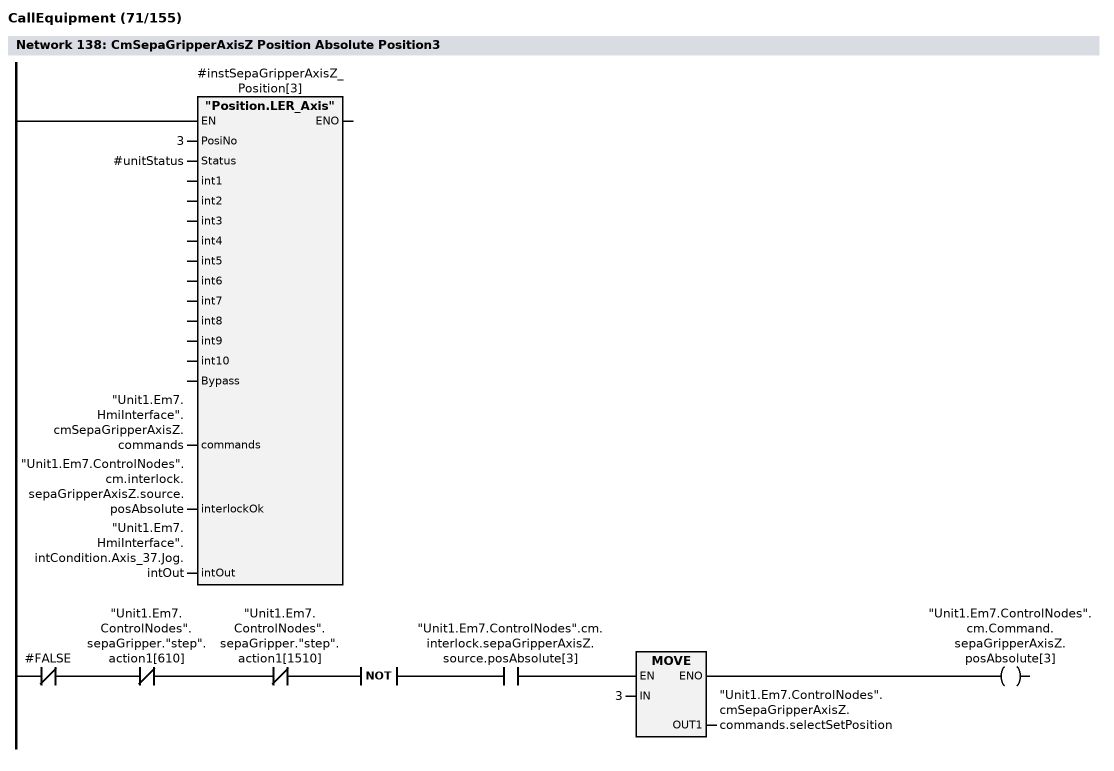
   RUNG wire#powerrail
      #instSepaGripperAxisZ_Position[3](PosiNo := 3, Status := #unitStatus, int1 :=, int2 :=, int3 :=, int4 :=, int5 :=, int6 :=, int7 :=, int8 :=, int9 :=, int10 :=, Bypass :=, commands := "Unit1.Em7.HmiInterface".cmSepaGripperAxisZ.commands, interlockOk := "Unit1.Em7.ControlNodes".cm.interlock.sepaGripperAxisZ.source.posAbsolute, intOut := "Unit1.Em7.HmiInterface".intCondition.Axis_37.Jog.intOut)
   END_RUNG
   RUNG wire#powerrail
      I_Contact( #FALSE )
      I_Contact( "Unit1.Em7.ControlNodes".sepaGripper."step".action1[610] )
      I_Contact( "Unit1.Em7.ControlNodes".sepaGripper."step".action1[1510] )
      Not()
      Contact( "Unit1.Em7.ControlNodes".cm.interlock.sepaGripperAxisZ.source.posAbsolute[3] )
      Move(in := 3, out1 => "Unit1.Em7.ControlNodes".cmSepaGripperAxisZ.commands.selectSetPosition)
      Coil( "Unit1.Em7.ControlNodes".cm.Command.sepaGripperAxisZ.posAbsolute[3] )
   END_RUNG
   // the same network as SCL:
   #instSepaGripperAxisZ_Position[3](PosiNo := 3,   // "Position.LER_Axis"
                           Status := #unitStatus,
                           commands := "Unit1.Em7.HmiInterface".cmSepaGripperAxisZ.commands,
                           interlockOk := "Unit1.Em7.ControlNodes".cm.interlock.sepaGripperAxisZ.source.posAbsolute,
                           intOut := "Unit1.Em7.HmiInterface".intCondition.Axis_37.Jog.intOut);
   #_w1 := NOT (NOT #FALSE AND NOT "Unit1.Em7.ControlNodes".sepaGripper."step".action1[610] AND NOT "Unit1.Em7.ControlNodes".sepaGripper."step".action1[1510]) AND "Unit1.Em7.ControlNodes".cm.interlock.sepaGripperAxisZ.source.posAbsolute[3];
   IF #_w1 THEN "Unit1.Em7.ControlNodes".cmSepaGripperAxisZ.commands.selectSetPosition := 3; END_IF;
   "Unit1.Em7.ControlNodes".cm.Command.sepaGripperAxisZ.posAbsolute[3] := #_w1;
END_REGION

REGION Network 139: CmSepaGripperAxisZ Position Absolute Position4
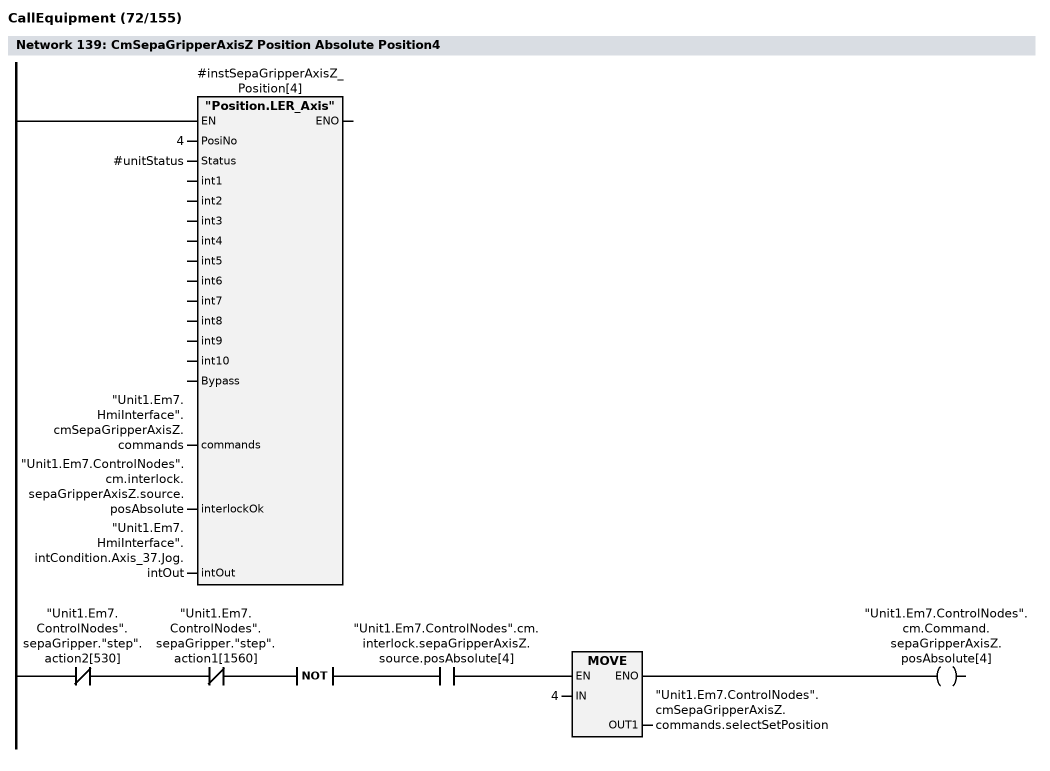
   RUNG wire#powerrail
      #instSepaGripperAxisZ_Position[4](PosiNo := 4, Status := #unitStatus, int1 :=, int2 :=, int3 :=, int4 :=, int5 :=, int6 :=, int7 :=, int8 :=, int9 :=, int10 :=, Bypass :=, commands := "Unit1.Em7.HmiInterface".cmSepaGripperAxisZ.commands, interlockOk := "Unit1.Em7.ControlNodes".cm.interlock.sepaGripperAxisZ.source.posAbsolute, intOut := "Unit1.Em7.HmiInterface".intCondition.Axis_37.Jog.intOut)
   END_RUNG
   RUNG wire#powerrail
      I_Contact( "Unit1.Em7.ControlNodes".sepaGripper."step".action2[530] )
      I_Contact( "Unit1.Em7.ControlNodes".sepaGripper."step".action1[1560] )
      Not()
      Contact( "Unit1.Em7.ControlNodes".cm.interlock.sepaGripperAxisZ.source.posAbsolute[4] )
      Move(in := 4, out1 => "Unit1.Em7.ControlNodes".cmSepaGripperAxisZ.commands.selectSetPosition)
      Coil( "Unit1.Em7.ControlNodes".cm.Command.sepaGripperAxisZ.posAbsolute[4] )
   END_RUNG
   // the same network as SCL:
   #instSepaGripperAxisZ_Position[4](PosiNo := 4,   // "Position.LER_Axis"
                           Status := #unitStatus,
                           commands := "Unit1.Em7.HmiInterface".cmSepaGripperAxisZ.commands,
                           interlockOk := "Unit1.Em7.ControlNodes".cm.interlock.sepaGripperAxisZ.source.posAbsolute,
                           intOut := "Unit1.Em7.HmiInterface".intCondition.Axis_37.Jog.intOut);
   #_w1 := NOT (NOT "Unit1.Em7.ControlNodes".sepaGripper."step".action2[530] AND NOT "Unit1.Em7.ControlNodes".sepaGripper."step".action1[1560]) AND "Unit1.Em7.ControlNodes".cm.interlock.sepaGripperAxisZ.source.posAbsolute[4];
   IF #_w1 THEN "Unit1.Em7.ControlNodes".cmSepaGripperAxisZ.commands.selectSetPosition := 4; END_IF;
   "Unit1.Em7.ControlNodes".cm.Command.sepaGripperAxisZ.posAbsolute[4] := #_w1;
END_REGION

REGION Network 140: CmSepaGripperAxisZ Position Absolute Position5
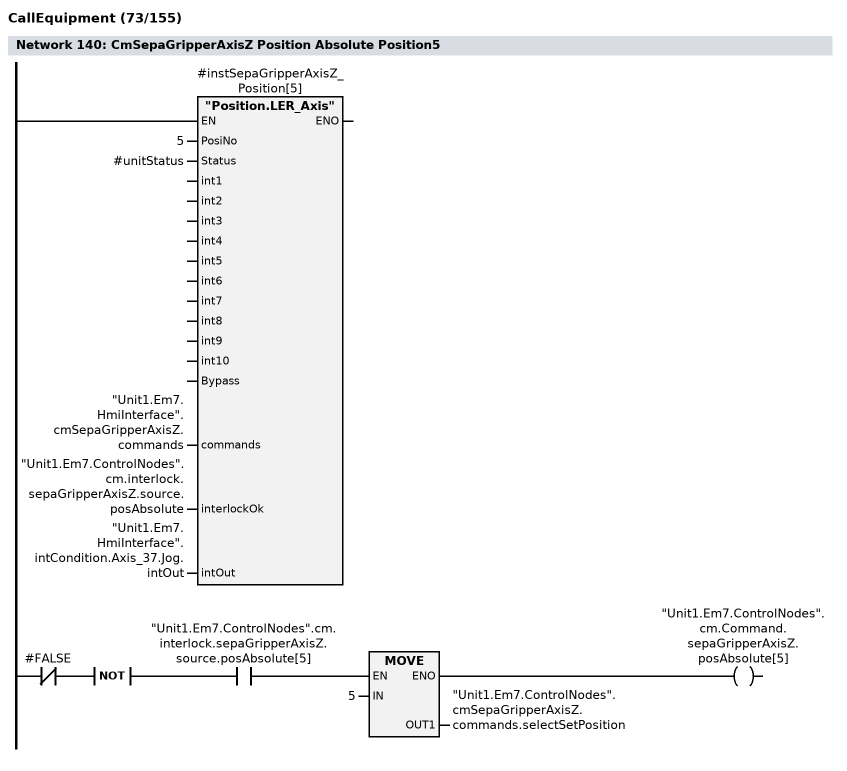
   RUNG wire#powerrail
      #instSepaGripperAxisZ_Position[5](PosiNo := 5, Status := #unitStatus, int1 :=, int2 :=, int3 :=, int4 :=, int5 :=, int6 :=, int7 :=, int8 :=, int9 :=, int10 :=, Bypass :=, commands := "Unit1.Em7.HmiInterface".cmSepaGripperAxisZ.commands, interlockOk := "Unit1.Em7.ControlNodes".cm.interlock.sepaGripperAxisZ.source.posAbsolute, intOut := "Unit1.Em7.HmiInterface".intCondition.Axis_37.Jog.intOut)
   END_RUNG
   RUNG wire#powerrail
      I_Contact( #FALSE )
      Not()
      Contact( "Unit1.Em7.ControlNodes".cm.interlock.sepaGripperAxisZ.source.posAbsolute[5] )
      Move(in := 5, out1 => "Unit1.Em7.ControlNodes".cmSepaGripperAxisZ.commands.selectSetPosition)
      Coil( "Unit1.Em7.ControlNodes".cm.Command.sepaGripperAxisZ.posAbsolute[5] )
   END_RUNG
   // the same network as SCL:
   #instSepaGripperAxisZ_Position[5](PosiNo := 5,   // "Position.LER_Axis"
                           Status := #unitStatus,
                           commands := "Unit1.Em7.HmiInterface".cmSepaGripperAxisZ.commands,
                           interlockOk := "Unit1.Em7.ControlNodes".cm.interlock.sepaGripperAxisZ.source.posAbsolute,
                           intOut := "Unit1.Em7.HmiInterface".intCondition.Axis_37.Jog.intOut);
   #_w1 := NOT (NOT #FALSE) AND "Unit1.Em7.ControlNodes".cm.interlock.sepaGripperAxisZ.source.posAbsolute[5];
   IF #_w1 THEN "Unit1.Em7.ControlNodes".cmSepaGripperAxisZ.commands.selectSetPosition := 5; END_IF;
   "Unit1.Em7.ControlNodes".cm.Command.sepaGripperAxisZ.posAbsolute[5] := #_w1;
END_REGION

REGION Network 141: CmSepaGripperAxisZ Position Absolute Position6
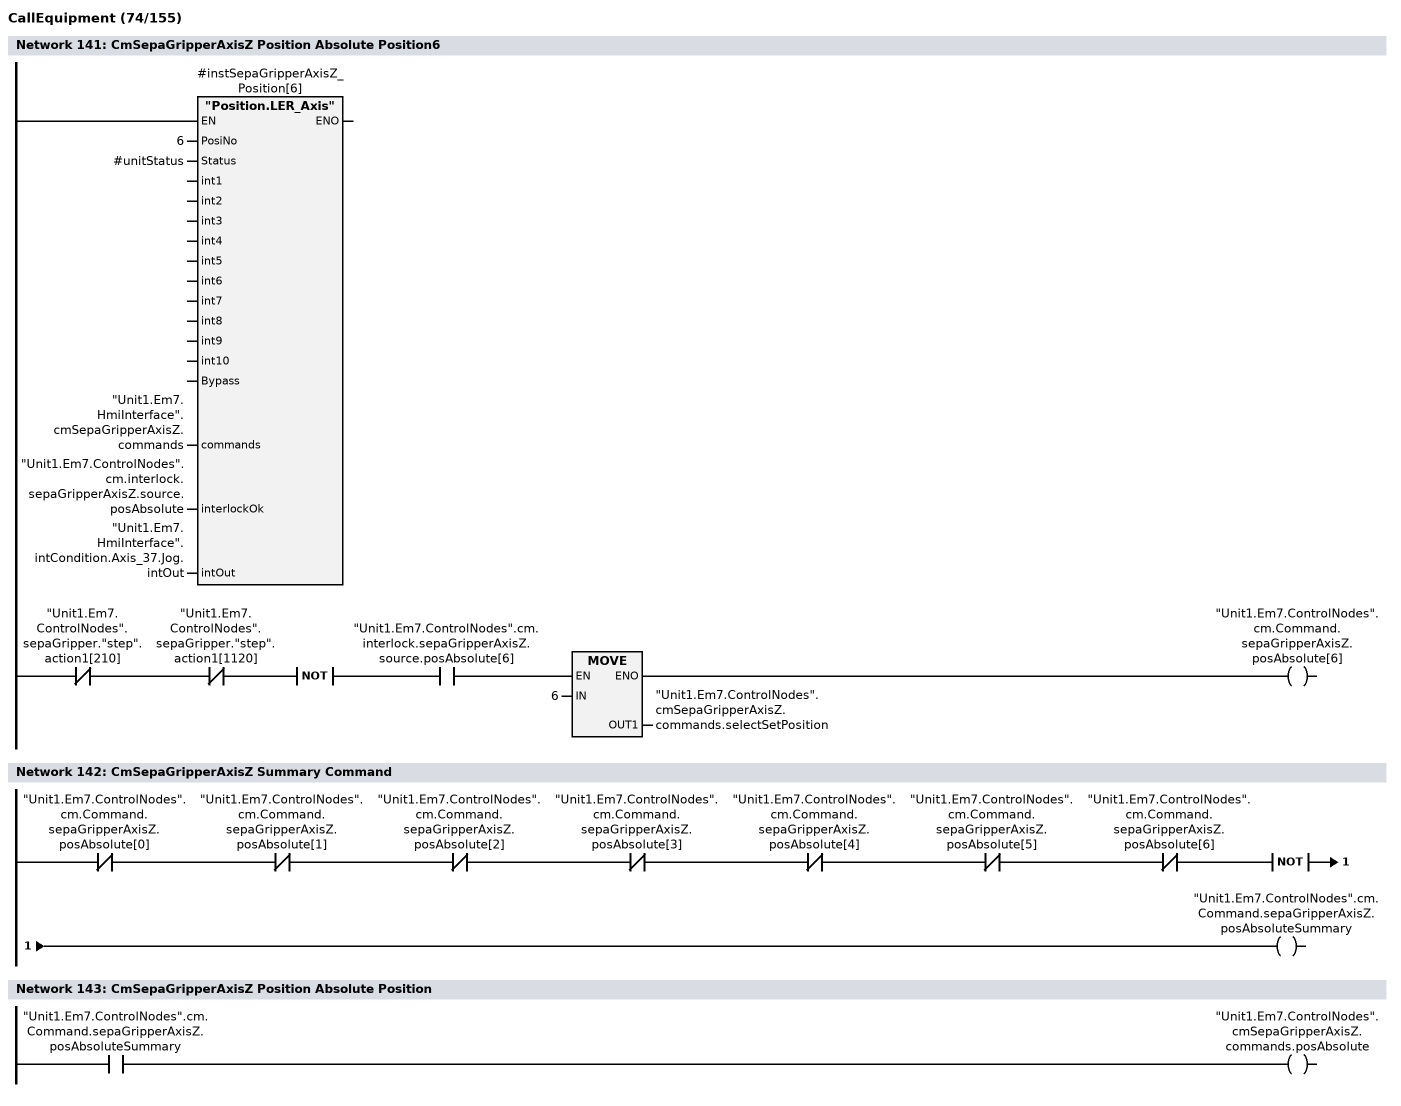
   RUNG wire#powerrail
      #instSepaGripperAxisZ_Position[6](PosiNo := 6, Status := #unitStatus, int1 :=, int2 :=, int3 :=, int4 :=, int5 :=, int6 :=, int7 :=, int8 :=, int9 :=, int10 :=, Bypass :=, commands := "Unit1.Em7.HmiInterface".cmSepaGripperAxisZ.commands, interlockOk := "Unit1.Em7.ControlNodes".cm.interlock.sepaGripperAxisZ.source.posAbsolute, intOut := "Unit1.Em7.HmiInterface".intCondition.Axis_37.Jog.intOut)
   END_RUNG
   RUNG wire#powerrail
      I_Contact( "Unit1.Em7.ControlNodes".sepaGripper."step".action1[210] )
      I_Contact( "Unit1.Em7.ControlNodes".sepaGripper."step".action1[1120] )
      Not()
      Contact( "Unit1.Em7.ControlNodes".cm.interlock.sepaGripperAxisZ.source.posAbsolute[6] )
      Move(in := 6, out1 => "Unit1.Em7.ControlNodes".cmSepaGripperAxisZ.commands.selectSetPosition)
      Coil( "Unit1.Em7.ControlNodes".cm.Command.sepaGripperAxisZ.posAbsolute[6] )
   END_RUNG
   // the same network as SCL:
   #instSepaGripperAxisZ_Position[6](PosiNo := 6,   // "Position.LER_Axis"
                           Status := #unitStatus,
                           commands := "Unit1.Em7.HmiInterface".cmSepaGripperAxisZ.commands,
                           interlockOk := "Unit1.Em7.ControlNodes".cm.interlock.sepaGripperAxisZ.source.posAbsolute,
                           intOut := "Unit1.Em7.HmiInterface".intCondition.Axis_37.Jog.intOut);
   #_w1 := NOT (NOT "Unit1.Em7.ControlNodes".sepaGripper."step".action1[210] AND NOT "Unit1.Em7.ControlNodes".sepaGripper."step".action1[1120]) AND "Unit1.Em7.ControlNodes".cm.interlock.sepaGripperAxisZ.source.posAbsolute[6];
   IF #_w1 THEN "Unit1.Em7.ControlNodes".cmSepaGripperAxisZ.commands.selectSetPosition := 6; END_IF;
   "Unit1.Em7.ControlNodes".cm.Command.sepaGripperAxisZ.posAbsolute[6] := #_w1;
END_REGION

REGION Network 142: CmSepaGripperAxisZ Summary Command
   RUNG wire#powerrail
      I_Contact( "Unit1.Em7.ControlNodes".cm.Command.sepaGripperAxisZ.posAbsolute[0] )
      I_Contact( "Unit1.Em7.ControlNodes".cm.Command.sepaGripperAxisZ.posAbsolute[1] )
      I_Contact( "Unit1.Em7.ControlNodes".cm.Command.sepaGripperAxisZ.posAbsolute[2] )
      I_Contact( "Unit1.Em7.ControlNodes".cm.Command.sepaGripperAxisZ.posAbsolute[3] )
      I_Contact( "Unit1.Em7.ControlNodes".cm.Command.sepaGripperAxisZ.posAbsolute[4] )
      I_Contact( "Unit1.Em7.ControlNodes".cm.Command.sepaGripperAxisZ.posAbsolute[5] )
      I_Contact( "Unit1.Em7.ControlNodes".cm.Command.sepaGripperAxisZ.posAbsolute[6] )
      Not()
      Coil( "Unit1.Em7.ControlNodes".cm.Command.sepaGripperAxisZ.posAbsoluteSummary )
   END_RUNG
   // the same network as SCL:
   "Unit1.Em7.ControlNodes".cm.Command.sepaGripperAxisZ.posAbsoluteSummary := NOT (NOT "Unit1.Em7.ControlNodes".cm.Command.sepaGripperAxisZ.posAbsolute[0] AND NOT "Unit1.Em7.ControlNodes".cm.Command.sepaGripperAxisZ.posAbsolute[1] AND NOT "Unit1.Em7.ControlNodes".cm.Command.sepaGripperAxisZ.posAbsolute[2] AND NOT "Unit1.Em7.ControlNodes".cm.Command.sepaGripperAxisZ.posAbsolute[3] AND NOT "Unit1.Em7.ControlNodes".cm.Command.sepaGripperAxisZ.posAbsolute[4] AND NOT "Unit1.Em7.ControlNodes".cm.Command.sepaGripperAxisZ.posAbsolute[5] AND NOT "Unit1.Em7.ControlNodes".cm.Command.sepaGripperAxisZ.posAbsolute[6]);
END_REGION

REGION Network 143: CmSepaGripperAxisZ Position Absolute Position
   RUNG wire#powerrail
      Contact( "Unit1.Em7.ControlNodes".cm.Command.sepaGripperAxisZ.posAbsoluteSummary )
      Coil( "Unit1.Em7.ControlNodes".cmSepaGripperAxisZ.commands.posAbsolute )
   END_RUNG
   // the same network as SCL:
   "Unit1.Em7.ControlNodes".cmSepaGripperAxisZ.commands.posAbsolute := "Unit1.Em7.ControlNodes".cm.Command.sepaGripperAxisZ.posAbsoluteSummary;
END_REGION

REGION Network 144: CmSepaGripperAxisZ Interlock Summary
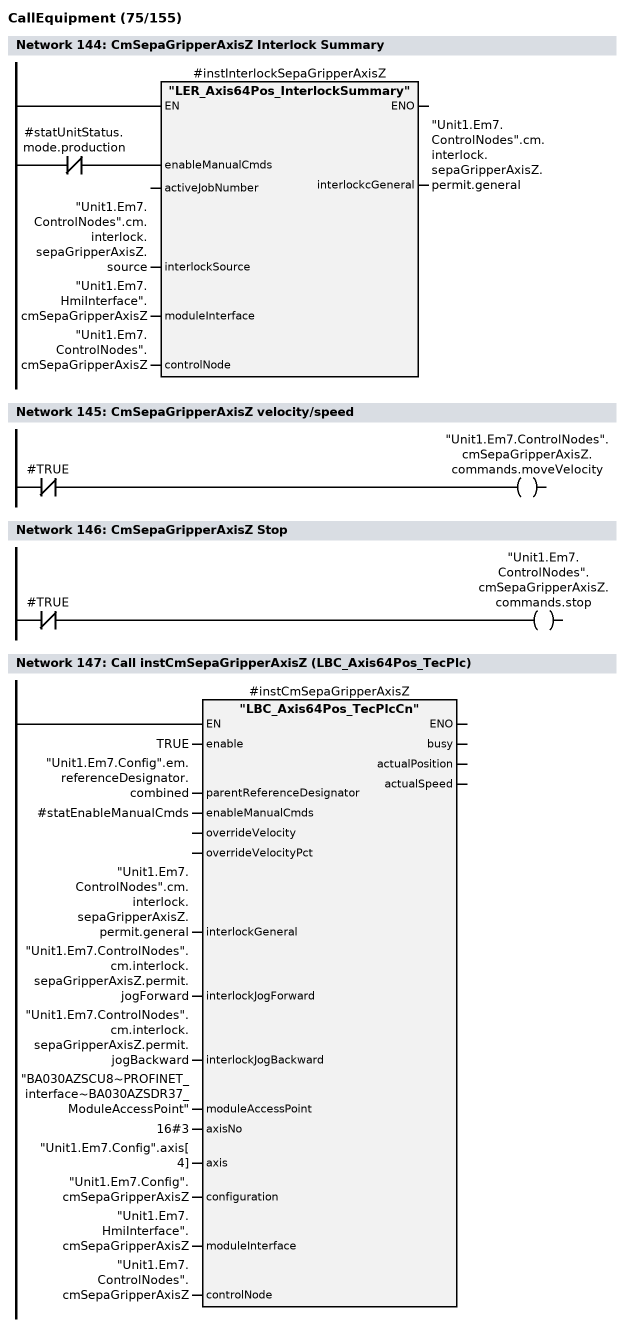
   RUNG wire#powerrail
      #instInterlockSepaGripperAxisZ(enableManualCmds := wire#w1, activeJobNumber :=, interlockSource := "Unit1.Em7.ControlNodes".cm.interlock.sepaGripperAxisZ.source, moduleInterface := "Unit1.Em7.HmiInterface".cmSepaGripperAxisZ, controlNode := "Unit1.Em7.ControlNodes".cmSepaGripperAxisZ, interlockcGeneral => "Unit1.Em7.ControlNodes".cm.interlock.sepaGripperAxisZ.permit.general)
   END_RUNG
   RUNG wire#powerrail
      I_Contact( #statUnitStatus.mode.production )
   END_RUNG wire#w1
   // the same network as SCL:
   #instInterlockSepaGripperAxisZ(enableManualCmds := NOT #statUnitStatus.mode.production,   // "LER_Axis64Pos_InterlockSummary"
                           interlockSource := "Unit1.Em7.ControlNodes".cm.interlock.sepaGripperAxisZ.source,
                           moduleInterface := "Unit1.Em7.HmiInterface".cmSepaGripperAxisZ,
                           controlNode := "Unit1.Em7.ControlNodes".cmSepaGripperAxisZ,
                           interlockcGeneral => "Unit1.Em7.ControlNodes".cm.interlock.sepaGripperAxisZ.permit.general);
END_REGION

REGION Network 145: CmSepaGripperAxisZ velocity/speed
   RUNG wire#powerrail
      I_Contact( #TRUE )
      Coil( "Unit1.Em7.ControlNodes".cmSepaGripperAxisZ.commands.moveVelocity )
   END_RUNG
   // the same network as SCL:
   "Unit1.Em7.ControlNodes".cmSepaGripperAxisZ.commands.moveVelocity := NOT #TRUE;
END_REGION

REGION Network 146: CmSepaGripperAxisZ Stop
   RUNG wire#powerrail
      I_Contact( #TRUE )
      Coil( "Unit1.Em7.ControlNodes".cmSepaGripperAxisZ.commands.stop )
   END_RUNG
   // the same network as SCL:
   "Unit1.Em7.ControlNodes".cmSepaGripperAxisZ.commands.stop := NOT #TRUE;
END_REGION

REGION Network 147: Call instCmSepaGripperAxisZ (LBC_Axis64Pos_TecPlc)
   RUNG wire#powerrail
      #instCmSepaGripperAxisZ(enable := TRUE, parentReferenceDesignator := "Unit1.Em7.Config".em.referenceDesignator.combined, enableManualCmds := #statEnableManualCmds, overrideVelocity :=, overrideVelocityPct :=, interlockGeneral := "Unit1.Em7.ControlNodes".cm.interlock.sepaGripperAxisZ.permit.general, interlockJogForward := "Unit1.Em7.ControlNodes".cm.interlock.sepaGripperAxisZ.permit.jogForward, interlockJogBackward := "Unit1.Em7.ControlNodes".cm.interlock.sepaGripperAxisZ.permit.jogBackward, moduleAccessPoint := "BA030AZSCU8~PROFINET_interface~BA030AZSDR37_ModuleAccessPoint", axisNo := 16#3, axis := "Unit1.Em7.Config".axis[4], configuration := "Unit1.Em7.Config".cmSepaGripperAxisZ, moduleInterface := "Unit1.Em7.HmiInterface".cmSepaGripperAxisZ, controlNode := "Unit1.Em7.ControlNodes".cmSepaGripperAxisZ, busy =>, actualPosition =>, actualSpeed =>)
   END_RUNG
   // the same network as SCL:
   #instCmSepaGripperAxisZ(enable := TRUE,   // "LBC_Axis64Pos_TecPlcCn"
                           parentReferenceDesignator := "Unit1.Em7.Config".em.referenceDesignator.combined,
                           enableManualCmds := #statEnableManualCmds,
                           interlockGeneral := "Unit1.Em7.ControlNodes".cm.interlock.sepaGripperAxisZ.permit.general,
                           interlockJogForward := "Unit1.Em7.ControlNodes".cm.interlock.sepaGripperAxisZ.permit.jogForward,
                           interlockJogBackward := "Unit1.Em7.ControlNodes".cm.interlock.sepaGripperAxisZ.permit.jogBackward,
                           moduleAccessPoint := "BA030AZSCU8~PROFINET_interface~BA030AZSDR37_ModuleAccessPoint",
                           axisNo := 16#3,
                           axis := "Unit1.Em7.Config".axis[4],
                           configuration := "Unit1.Em7.Config".cmSepaGripperAxisZ,
                           moduleInterface := "Unit1.Em7.HmiInterface".cmSepaGripperAxisZ,
                           controlNode := "Unit1.Em7.ControlNodes".cmSepaGripperAxisZ);
END_REGION

REGION Network 148: CmSepaGripperAxisZ SoftCam
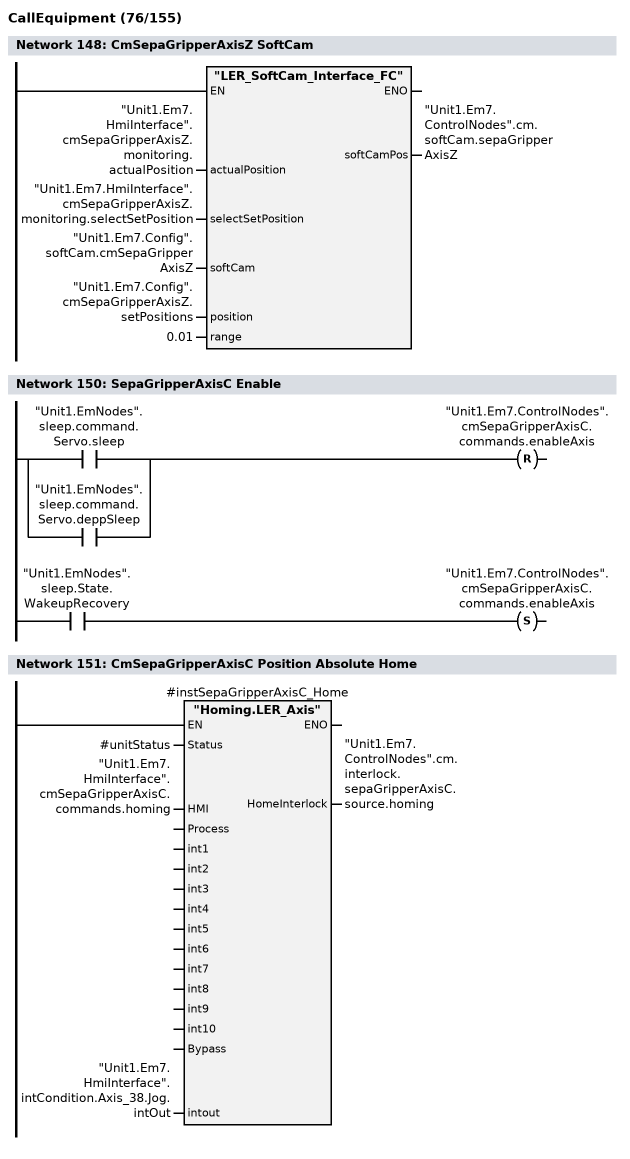
   RUNG wire#powerrail
      "LER_SoftCam_Interface_FC"(actualPosition := "Unit1.Em7.HmiInterface".cmSepaGripperAxisZ.monitoring.actualPosition, selectSetPosition := "Unit1.Em7.HmiInterface".cmSepaGripperAxisZ.monitoring.selectSetPosition, softCam := "Unit1.Em7.Config".softCam.cmSepaGripperAxisZ, position := "Unit1.Em7.Config".cmSepaGripperAxisZ.setPositions, range := 0.01, softCamPos => "Unit1.Em7.ControlNodes".cm.softCam.sepaGripperAxisZ)
   END_RUNG
   // the same network as SCL:
   "LER_SoftCam_Interface_FC"(actualPosition := "Unit1.Em7.HmiInterface".cmSepaGripperAxisZ.monitoring.actualPosition,
                           selectSetPosition := "Unit1.Em7.HmiInterface".cmSepaGripperAxisZ.monitoring.selectSetPosition,
                           softCam := "Unit1.Em7.Config".softCam.cmSepaGripperAxisZ,
                           position := "Unit1.Em7.Config".cmSepaGripperAxisZ.setPositions,
                           range := 0.01,
                           softCamPos => "Unit1.Em7.ControlNodes".cm.softCam.sepaGripperAxisZ);
END_REGION

REGION Network 150: SepaGripperAxisC Enable
   RUNG wire#powerrail
      Contact( "Unit1.EmNodes".sleep.command.Servo.sleep )
      wire#w1
      R_Coil( "Unit1.Em7.ControlNodes".cmSepaGripperAxisC.commands.enableAxis )
   END_RUNG
   RUNG wire#powerrail
      Contact( "Unit1.EmNodes".sleep.command.Servo.deppSleep )
   END_RUNG wire#w1
   RUNG wire#powerrail
      Contact( "Unit1.EmNodes".sleep.State.WakeupRecovery )
      S_Coil( "Unit1.Em7.ControlNodes".cmSepaGripperAxisC.commands.enableAxis )
   END_RUNG
   // the same network as SCL:
   IF "Unit1.EmNodes".sleep.command.Servo.sleep OR "Unit1.EmNodes".sleep.command.Servo.deppSleep THEN
       "Unit1.Em7.ControlNodes".cmSepaGripperAxisC.commands.enableAxis := FALSE;
   END_IF;
   IF "Unit1.EmNodes".sleep.State.WakeupRecovery THEN
       "Unit1.Em7.ControlNodes".cmSepaGripperAxisC.commands.enableAxis := TRUE;
   END_IF;
END_REGION

REGION Network 151: CmSepaGripperAxisC Position Absolute Home
   RUNG wire#powerrail
      #instSepaGripperAxisC_Home(Status := #unitStatus, HMI := "Unit1.Em7.HmiInterface".cmSepaGripperAxisC.commands.homing, Process :=, int1 :=, int2 :=, int3 :=, int4 :=, int5 :=, int6 :=, int7 :=, int8 :=, int9 :=, int10 :=, Bypass :=, intout := "Unit1.Em7.HmiInterface".intCondition.Axis_38.Jog.intOut, HomeInterlock => "Unit1.Em7.ControlNodes".cm.interlock.sepaGripperAxisC.source.homing)
   END_RUNG
   // the same network as SCL:
   #instSepaGripperAxisC_Home(Status := #unitStatus,   // "Homing.LER_Axis"
                           HMI := "Unit1.Em7.HmiInterface".cmSepaGripperAxisC.commands.homing,
                           intout := "Unit1.Em7.HmiInterface".intCondition.Axis_38.Jog.intOut,
                           HomeInterlock => "Unit1.Em7.ControlNodes".cm.interlock.sepaGripperAxisC.source.homing);
END_REGION

REGION Network 152: CmSepaGripperAxisC Position Absolute Jog
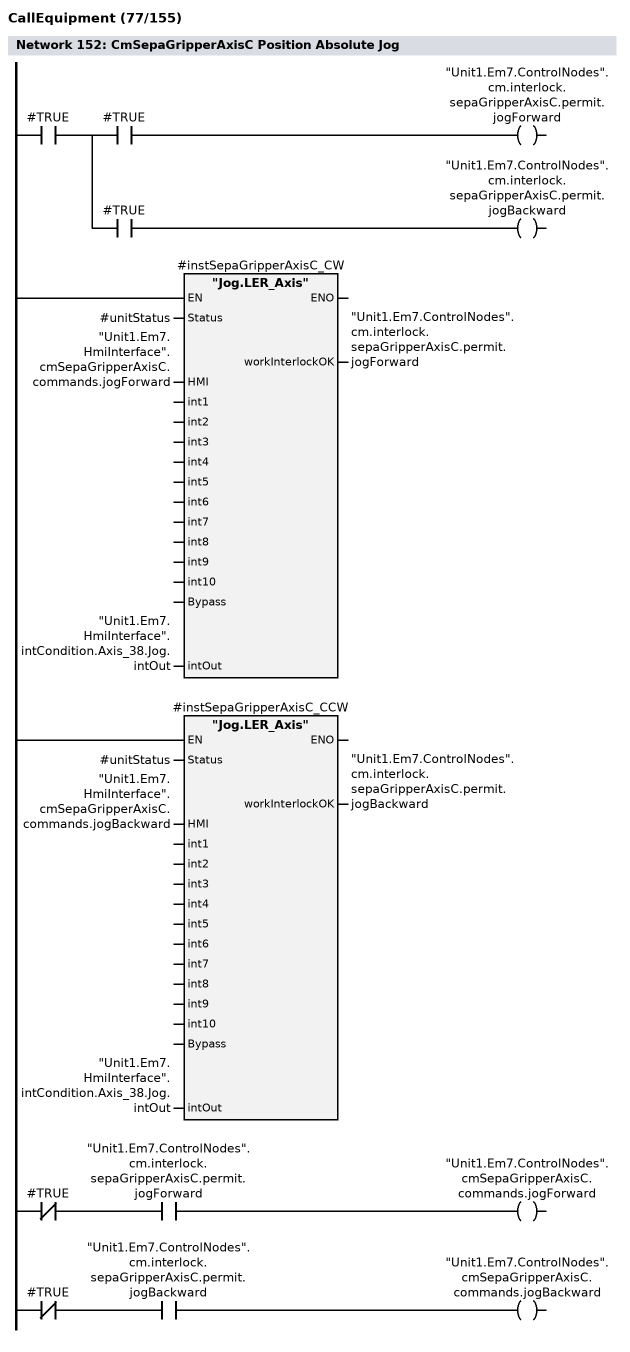
   RUNG wire#powerrail
      Contact( #TRUE )
      wire#w1
      Contact( #TRUE )
      Coil( "Unit1.Em7.ControlNodes".cm.interlock.sepaGripperAxisC.permit.jogForward )
   END_RUNG
   RUNG wire#w1
      Contact( #TRUE )
      Coil( "Unit1.Em7.ControlNodes".cm.interlock.sepaGripperAxisC.permit.jogBackward )
   END_RUNG
   RUNG wire#powerrail
      #instSepaGripperAxisC_CW(Status := #unitStatus, HMI := "Unit1.Em7.HmiInterface".cmSepaGripperAxisC.commands.jogForward, int1 :=, int2 :=, int3 :=, int4 :=, int5 :=, int6 :=, int7 :=, int8 :=, int9 :=, int10 :=, Bypass :=, intOut := "Unit1.Em7.HmiInterface".intCondition.Axis_38.Jog.intOut, workInterlockOK => "Unit1.Em7.ControlNodes".cm.interlock.sepaGripperAxisC.permit.jogForward)
   END_RUNG
   RUNG wire#powerrail
      #instSepaGripperAxisC_CCW(Status := #unitStatus, HMI := "Unit1.Em7.HmiInterface".cmSepaGripperAxisC.commands.jogBackward, int1 :=, int2 :=, int3 :=, int4 :=, int5 :=, int6 :=, int7 :=, int8 :=, int9 :=, int10 :=, Bypass :=, intOut := "Unit1.Em7.HmiInterface".intCondition.Axis_38.Jog.intOut, workInterlockOK => "Unit1.Em7.ControlNodes".cm.interlock.sepaGripperAxisC.permit.jogBackward)
   END_RUNG
   RUNG wire#powerrail
      I_Contact( #TRUE )
      Contact( "Unit1.Em7.ControlNodes".cm.interlock.sepaGripperAxisC.permit.jogForward )
      Coil( "Unit1.Em7.ControlNodes".cmSepaGripperAxisC.commands.jogForward )
   END_RUNG
   RUNG wire#powerrail
      I_Contact( #TRUE )
      Contact( "Unit1.Em7.ControlNodes".cm.interlock.sepaGripperAxisC.permit.jogBackward )
      Coil( "Unit1.Em7.ControlNodes".cmSepaGripperAxisC.commands.jogBackward )
   END_RUNG
   // the same network as SCL:
   "Unit1.Em7.ControlNodes".cm.interlock.sepaGripperAxisC.permit.jogForward := #TRUE AND #TRUE;
   "Unit1.Em7.ControlNodes".cm.interlock.sepaGripperAxisC.permit.jogBackward := #TRUE AND #TRUE;
   #instSepaGripperAxisC_CW(Status := #unitStatus,   // "Jog.LER_Axis"
                           HMI := "Unit1.Em7.HmiInterface".cmSepaGripperAxisC.commands.jogForward,
                           intOut := "Unit1.Em7.HmiInterface".intCondition.Axis_38.Jog.intOut,
                           workInterlockOK => "Unit1.Em7.ControlNodes".cm.interlock.sepaGripperAxisC.permit.jogForward);
   #instSepaGripperAxisC_CCW(Status := #unitStatus,   // "Jog.LER_Axis"
                           HMI := "Unit1.Em7.HmiInterface".cmSepaGripperAxisC.commands.jogBackward,
                           intOut := "Unit1.Em7.HmiInterface".intCondition.Axis_38.Jog.intOut,
                           workInterlockOK => "Unit1.Em7.ControlNodes".cm.interlock.sepaGripperAxisC.permit.jogBackward);
   "Unit1.Em7.ControlNodes".cmSepaGripperAxisC.commands.jogForward := NOT #TRUE AND "Unit1.Em7.ControlNodes".cm.interlock.sepaGripperAxisC.permit.jogForward;
   "Unit1.Em7.ControlNodes".cmSepaGripperAxisC.commands.jogBackward := NOT #TRUE AND "Unit1.Em7.ControlNodes".cm.interlock.sepaGripperAxisC.permit.jogBackward;
END_REGION

REGION Network 153: CmSepaGripperAxisC Position Absolute Position0
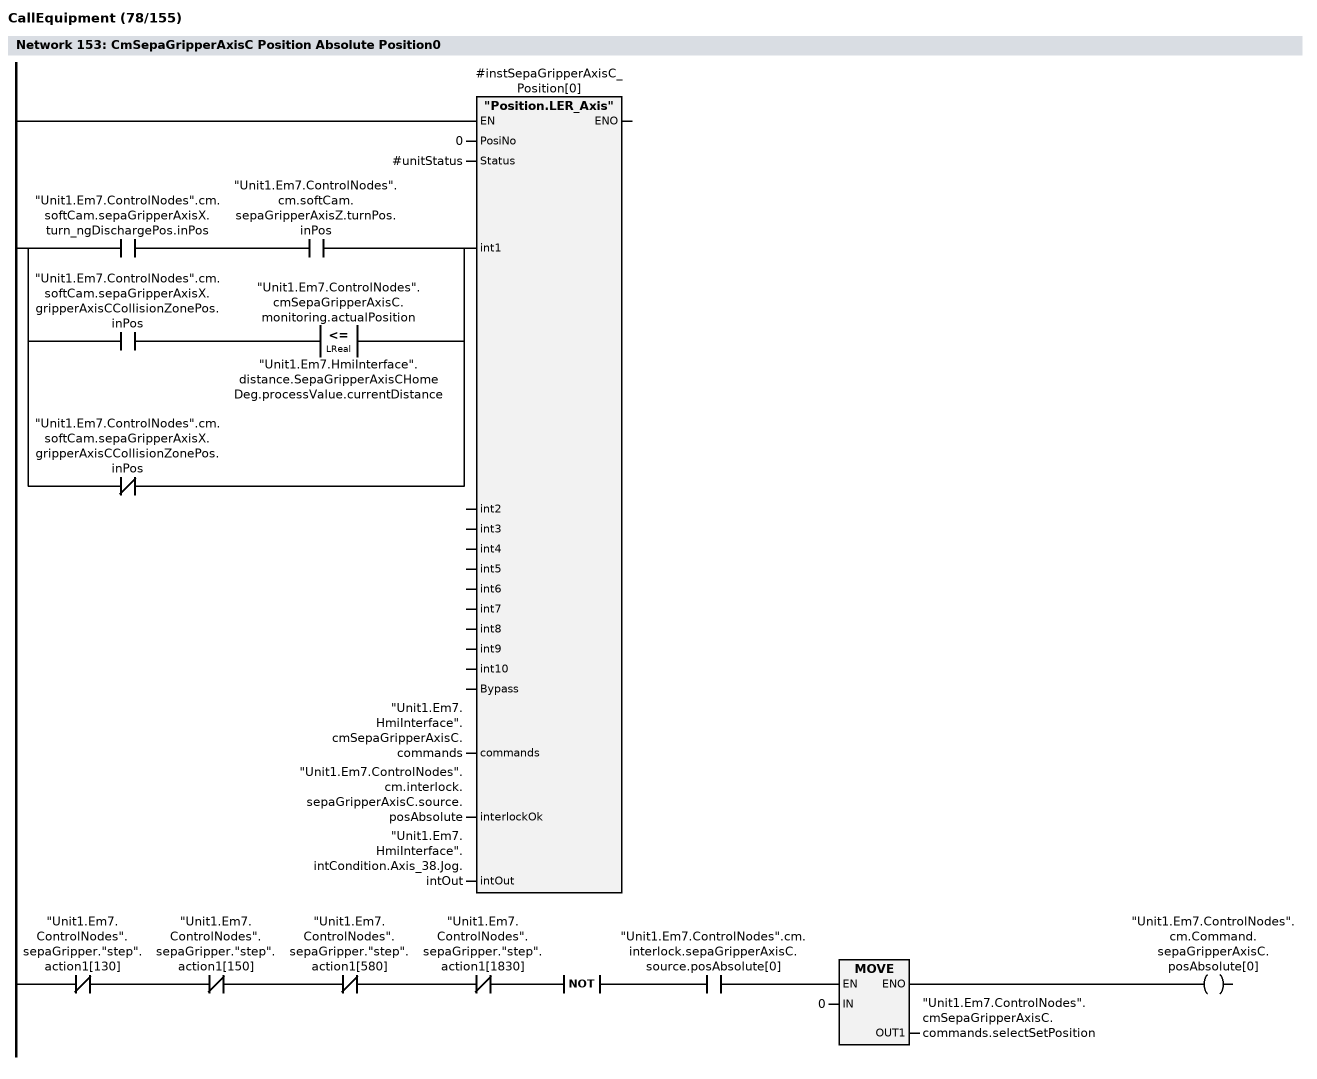
   RUNG wire#powerrail
      #instSepaGripperAxisC_Position[0](int1 := wire#w1, PosiNo := 0, Status := #unitStatus, int2 :=, int3 :=, int4 :=, int5 :=, int6 :=, int7 :=, int8 :=, int9 :=, int10 :=, Bypass :=, commands := "Unit1.Em7.HmiInterface".cmSepaGripperAxisC.commands, interlockOk := "Unit1.Em7.ControlNodes".cm.interlock.sepaGripperAxisC.source.posAbsolute, intOut := "Unit1.Em7.HmiInterface".intCondition.Axis_38.Jog.intOut)
   END_RUNG
   RUNG wire#powerrail
      Contact( "Unit1.Em7.ControlNodes".cm.softCam.sepaGripperAxisX.turn_ngDischargePos.inPos )
      Contact( "Unit1.Em7.ControlNodes".cm.softCam.sepaGripperAxisZ.turnPos.inPos )
   END_RUNG wire#w1
   RUNG wire#powerrail
      Contact( "Unit1.Em7.ControlNodes".cm.softCam.sepaGripperAxisX.gripperAxisCCollisionZonePos.inPos )
      { S7_Templates := "SrcType := LReal" } LE_Contact(in1 := "Unit1.Em7.ControlNodes".cmSepaGripperAxisC.monitoring.actualPosition, in2 := "Unit1.Em7.HmiInterface".distance.SepaGripperAxisCHomeDeg.processValue.currentDistance)
   END_RUNG wire#w1
   RUNG wire#powerrail
      I_Contact( "Unit1.Em7.ControlNodes".cm.softCam.sepaGripperAxisX.gripperAxisCCollisionZonePos.inPos )
   END_RUNG wire#w1
   RUNG wire#powerrail
      I_Contact( "Unit1.Em7.ControlNodes".sepaGripper."step".action1[130] )
      I_Contact( "Unit1.Em7.ControlNodes".sepaGripper."step".action1[150] )
      I_Contact( "Unit1.Em7.ControlNodes".sepaGripper."step".action1[580] )
      I_Contact( "Unit1.Em7.ControlNodes".sepaGripper."step".action1[1830] )
      Not()
      Contact( "Unit1.Em7.ControlNodes".cm.interlock.sepaGripperAxisC.source.posAbsolute[0] )
      Move(in := 0, out1 => "Unit1.Em7.ControlNodes".cmSepaGripperAxisC.commands.selectSetPosition)
      Coil( "Unit1.Em7.ControlNodes".cm.Command.sepaGripperAxisC.posAbsolute[0] )
   END_RUNG
   // the same network as SCL:
   #instSepaGripperAxisC_Position[0](PosiNo := 0,   // "Position.LER_Axis"
                           Status := #unitStatus,
                           int1 := ("Unit1.Em7.ControlNodes".cm.softCam.sepaGripperAxisX.turn_ngDischargePos.inPos AND "Unit1.Em7.ControlNodes".cm.softCam.sepaGripperAxisZ.turnPos.inPos) OR ("Unit1.Em7.ControlNodes".cm.softCam.sepaGripperAxisX.gripperAxisCCollisionZonePos.inPos AND ("Unit1.Em7.ControlNodes".cmSepaGripperAxisC.monitoring.actualPosition <= "Unit1.Em7.HmiInterface".distance.SepaGripperAxisCHomeDeg.processValue.currentDistance)) OR NOT "Unit1.Em7.ControlNodes".cm.softCam.sepaGripperAxisX.gripperAxisCCollisionZonePos.inPos,
                           commands := "Unit1.Em7.HmiInterface".cmSepaGripperAxisC.commands,
                           interlockOk := "Unit1.Em7.ControlNodes".cm.interlock.sepaGripperAxisC.source.posAbsolute,
                           intOut := "Unit1.Em7.HmiInterface".intCondition.Axis_38.Jog.intOut);
   #_w1 := NOT (NOT "Unit1.Em7.ControlNodes".sepaGripper."step".action1[130] AND NOT "Unit1.Em7.ControlNodes".sepaGripper."step".action1[150] AND NOT "Unit1.Em7.ControlNodes".sepaGripper."step".action1[580] AND NOT "Unit1.Em7.ControlNodes".sepaGripper."step".action1[1830]) AND "Unit1.Em7.ControlNodes".cm.interlock.sepaGripperAxisC.source.posAbsolute[0];
   IF #_w1 THEN "Unit1.Em7.ControlNodes".cmSepaGripperAxisC.commands.selectSetPosition := 0; END_IF;
   "Unit1.Em7.ControlNodes".cm.Command.sepaGripperAxisC.posAbsolute[0] := #_w1;
END_REGION

REGION Network 154: CmSepaGripperAxisC Position Absolute Position1
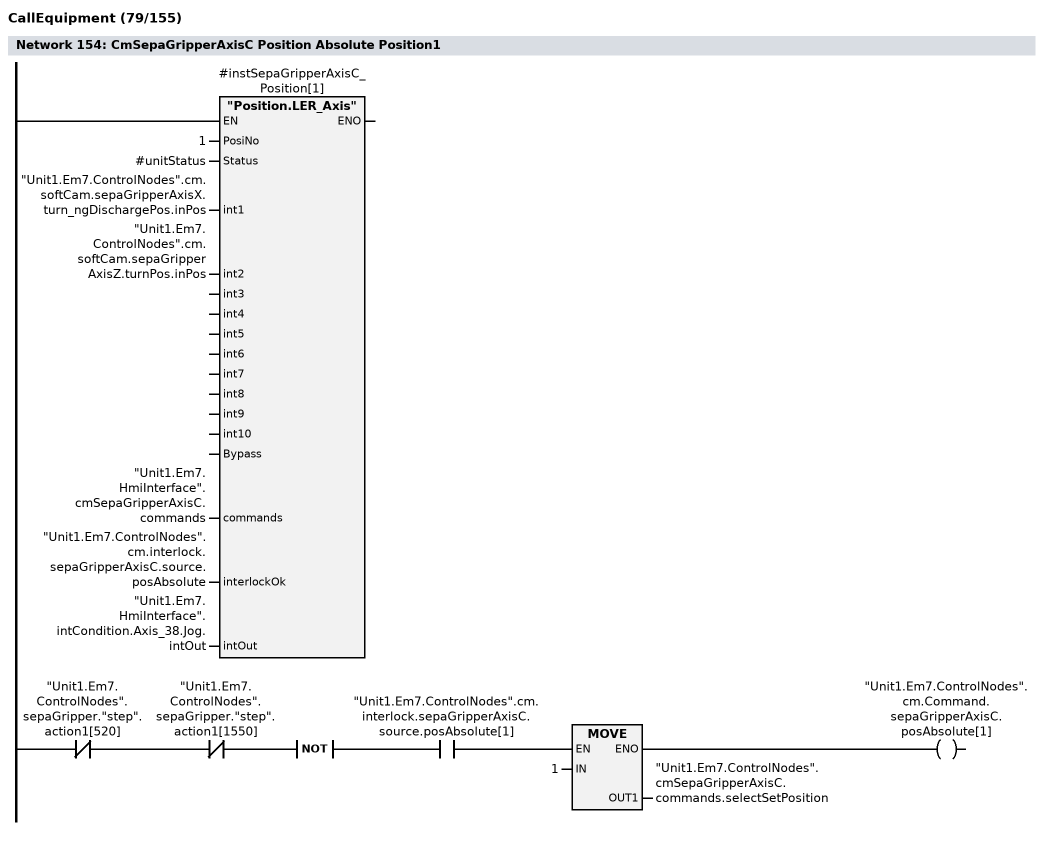
   RUNG wire#powerrail
      #instSepaGripperAxisC_Position[1](PosiNo := 1, Status := #unitStatus, int1 := "Unit1.Em7.ControlNodes".cm.softCam.sepaGripperAxisX.turn_ngDischargePos.inPos, int2 := "Unit1.Em7.ControlNodes".cm.softCam.sepaGripperAxisZ.turnPos.inPos, int3 :=, int4 :=, int5 :=, int6 :=, int7 :=, int8 :=, int9 :=, int10 :=, Bypass :=, commands := "Unit1.Em7.HmiInterface".cmSepaGripperAxisC.commands, interlockOk := "Unit1.Em7.ControlNodes".cm.interlock.sepaGripperAxisC.source.posAbsolute, intOut := "Unit1.Em7.HmiInterface".intCondition.Axis_38.Jog.intOut)
   END_RUNG
   RUNG wire#powerrail
      I_Contact( "Unit1.Em7.ControlNodes".sepaGripper."step".action1[520] )
      I_Contact( "Unit1.Em7.ControlNodes".sepaGripper."step".action1[1550] )
      Not()
      Contact( "Unit1.Em7.ControlNodes".cm.interlock.sepaGripperAxisC.source.posAbsolute[1] )
      Move(in := 1, out1 => "Unit1.Em7.ControlNodes".cmSepaGripperAxisC.commands.selectSetPosition)
      Coil( "Unit1.Em7.ControlNodes".cm.Command.sepaGripperAxisC.posAbsolute[1] )
   END_RUNG
   // the same network as SCL:
   #instSepaGripperAxisC_Position[1](PosiNo := 1,   // "Position.LER_Axis"
                           Status := #unitStatus,
                           int1 := "Unit1.Em7.ControlNodes".cm.softCam.sepaGripperAxisX.turn_ngDischargePos.inPos,
                           int2 := "Unit1.Em7.ControlNodes".cm.softCam.sepaGripperAxisZ.turnPos.inPos,
                           commands := "Unit1.Em7.HmiInterface".cmSepaGripperAxisC.commands,
                           interlockOk := "Unit1.Em7.ControlNodes".cm.interlock.sepaGripperAxisC.source.posAbsolute,
                           intOut := "Unit1.Em7.HmiInterface".intCondition.Axis_38.Jog.intOut);
   #_w1 := NOT (NOT "Unit1.Em7.ControlNodes".sepaGripper."step".action1[520] AND NOT "Unit1.Em7.ControlNodes".sepaGripper."step".action1[1550]) AND "Unit1.Em7.ControlNodes".cm.interlock.sepaGripperAxisC.source.posAbsolute[1];
   IF #_w1 THEN "Unit1.Em7.ControlNodes".cmSepaGripperAxisC.commands.selectSetPosition := 1; END_IF;
   "Unit1.Em7.ControlNodes".cm.Command.sepaGripperAxisC.posAbsolute[1] := #_w1;
END_REGION

REGION Network 155: CmSepaGripperAxisC Position Absolute Position2
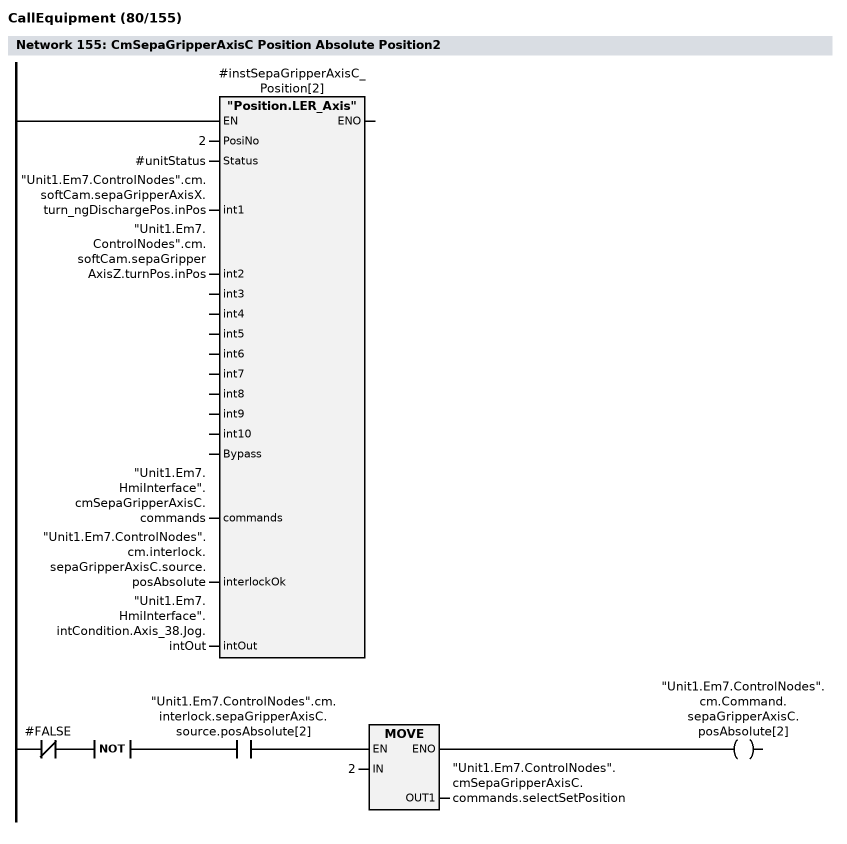
   RUNG wire#powerrail
      #instSepaGripperAxisC_Position[2](PosiNo := 2, Status := #unitStatus, int1 := "Unit1.Em7.ControlNodes".cm.softCam.sepaGripperAxisX.turn_ngDischargePos.inPos, int2 := "Unit1.Em7.ControlNodes".cm.softCam.sepaGripperAxisZ.turnPos.inPos, int3 :=, int4 :=, int5 :=, int6 :=, int7 :=, int8 :=, int9 :=, int10 :=, Bypass :=, commands := "Unit1.Em7.HmiInterface".cmSepaGripperAxisC.commands, interlockOk := "Unit1.Em7.ControlNodes".cm.interlock.sepaGripperAxisC.source.posAbsolute, intOut := "Unit1.Em7.HmiInterface".intCondition.Axis_38.Jog.intOut)
   END_RUNG
   RUNG wire#powerrail
      I_Contact( #FALSE )
      Not()
      Contact( "Unit1.Em7.ControlNodes".cm.interlock.sepaGripperAxisC.source.posAbsolute[2] )
      Move(in := 2, out1 => "Unit1.Em7.ControlNodes".cmSepaGripperAxisC.commands.selectSetPosition)
      Coil( "Unit1.Em7.ControlNodes".cm.Command.sepaGripperAxisC.posAbsolute[2] )
   END_RUNG
   // the same network as SCL:
   #instSepaGripperAxisC_Position[2](PosiNo := 2,   // "Position.LER_Axis"
                           Status := #unitStatus,
                           int1 := "Unit1.Em7.ControlNodes".cm.softCam.sepaGripperAxisX.turn_ngDischargePos.inPos,
                           int2 := "Unit1.Em7.ControlNodes".cm.softCam.sepaGripperAxisZ.turnPos.inPos,
                           commands := "Unit1.Em7.HmiInterface".cmSepaGripperAxisC.commands,
                           interlockOk := "Unit1.Em7.ControlNodes".cm.interlock.sepaGripperAxisC.source.posAbsolute,
                           intOut := "Unit1.Em7.HmiInterface".intCondition.Axis_38.Jog.intOut);
   #_w1 := NOT (NOT #FALSE) AND "Unit1.Em7.ControlNodes".cm.interlock.sepaGripperAxisC.source.posAbsolute[2];
   IF #_w1 THEN "Unit1.Em7.ControlNodes".cmSepaGripperAxisC.commands.selectSetPosition := 2; END_IF;
   "Unit1.Em7.ControlNodes".cm.Command.sepaGripperAxisC.posAbsolute[2] := #_w1;
END_REGION

REGION Network 156: CmSepaGripperAxisC Position Absolute Position3
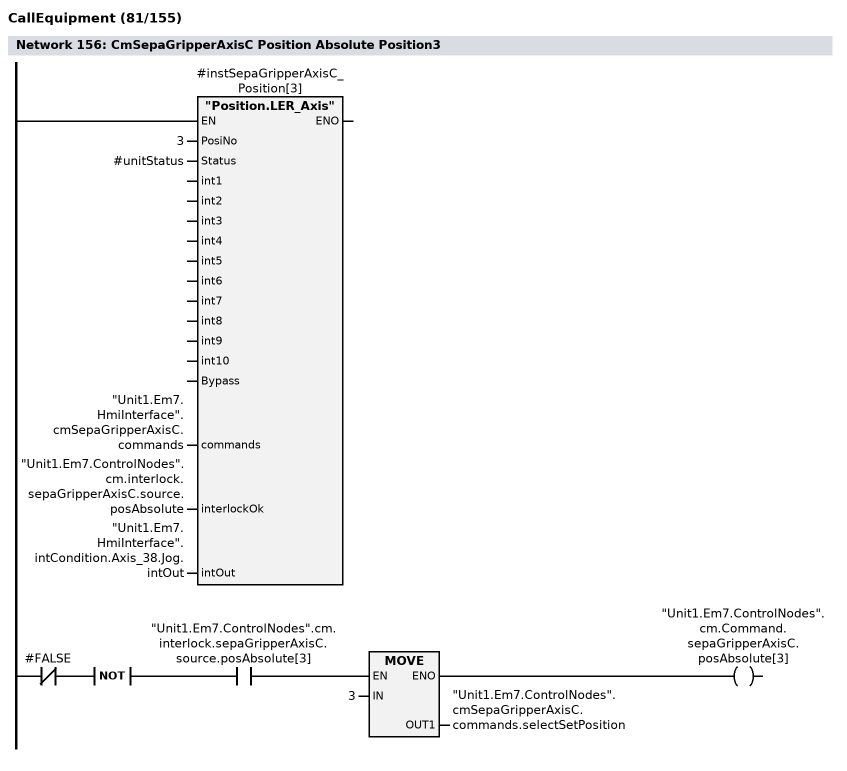
   RUNG wire#powerrail
      #instSepaGripperAxisC_Position[3](PosiNo := 3, Status := #unitStatus, int1 :=, int2 :=, int3 :=, int4 :=, int5 :=, int6 :=, int7 :=, int8 :=, int9 :=, int10 :=, Bypass :=, commands := "Unit1.Em7.HmiInterface".cmSepaGripperAxisC.commands, interlockOk := "Unit1.Em7.ControlNodes".cm.interlock.sepaGripperAxisC.source.posAbsolute, intOut := "Unit1.Em7.HmiInterface".intCondition.Axis_38.Jog.intOut)
   END_RUNG
   RUNG wire#powerrail
      I_Contact( #FALSE )
      Not()
      Contact( "Unit1.Em7.ControlNodes".cm.interlock.sepaGripperAxisC.source.posAbsolute[3] )
      Move(in := 3, out1 => "Unit1.Em7.ControlNodes".cmSepaGripperAxisC.commands.selectSetPosition)
      Coil( "Unit1.Em7.ControlNodes".cm.Command.sepaGripperAxisC.posAbsolute[3] )
   END_RUNG
   // the same network as SCL:
   #instSepaGripperAxisC_Position[3](PosiNo := 3,   // "Position.LER_Axis"
                           Status := #unitStatus,
                           commands := "Unit1.Em7.HmiInterface".cmSepaGripperAxisC.commands,
                           interlockOk := "Unit1.Em7.ControlNodes".cm.interlock.sepaGripperAxisC.source.posAbsolute,
                           intOut := "Unit1.Em7.HmiInterface".intCondition.Axis_38.Jog.intOut);
   #_w1 := NOT (NOT #FALSE) AND "Unit1.Em7.ControlNodes".cm.interlock.sepaGripperAxisC.source.posAbsolute[3];
   IF #_w1 THEN "Unit1.Em7.ControlNodes".cmSepaGripperAxisC.commands.selectSetPosition := 3; END_IF;
   "Unit1.Em7.ControlNodes".cm.Command.sepaGripperAxisC.posAbsolute[3] := #_w1;
END_REGION

REGION Network 157: CmSepaGripperAxisC Position Absolute Position4
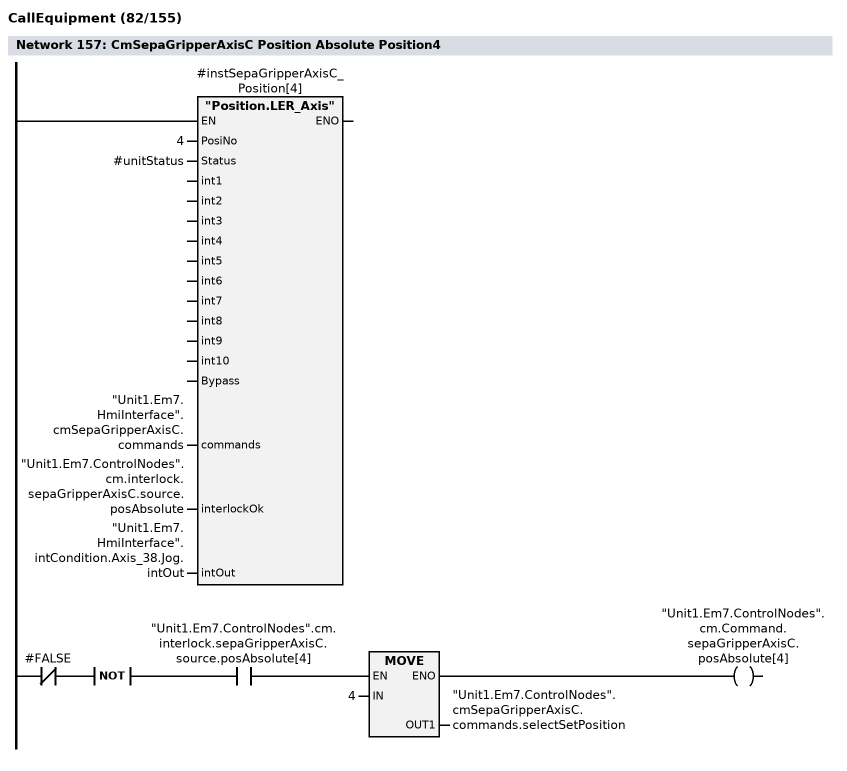
   RUNG wire#powerrail
      #instSepaGripperAxisC_Position[4](PosiNo := 4, Status := #unitStatus, int1 :=, int2 :=, int3 :=, int4 :=, int5 :=, int6 :=, int7 :=, int8 :=, int9 :=, int10 :=, Bypass :=, commands := "Unit1.Em7.HmiInterface".cmSepaGripperAxisC.commands, interlockOk := "Unit1.Em7.ControlNodes".cm.interlock.sepaGripperAxisC.source.posAbsolute, intOut := "Unit1.Em7.HmiInterface".intCondition.Axis_38.Jog.intOut)
   END_RUNG
   RUNG wire#powerrail
      I_Contact( #FALSE )
      Not()
      Contact( "Unit1.Em7.ControlNodes".cm.interlock.sepaGripperAxisC.source.posAbsolute[4] )
      Move(in := 4, out1 => "Unit1.Em7.ControlNodes".cmSepaGripperAxisC.commands.selectSetPosition)
      Coil( "Unit1.Em7.ControlNodes".cm.Command.sepaGripperAxisC.posAbsolute[4] )
   END_RUNG
   // the same network as SCL:
   #instSepaGripperAxisC_Position[4](PosiNo := 4,   // "Position.LER_Axis"
                           Status := #unitStatus,
                           commands := "Unit1.Em7.HmiInterface".cmSepaGripperAxisC.commands,
                           interlockOk := "Unit1.Em7.ControlNodes".cm.interlock.sepaGripperAxisC.source.posAbsolute,
                           intOut := "Unit1.Em7.HmiInterface".intCondition.Axis_38.Jog.intOut);
   #_w1 := NOT (NOT #FALSE) AND "Unit1.Em7.ControlNodes".cm.interlock.sepaGripperAxisC.source.posAbsolute[4];
   IF #_w1 THEN "Unit1.Em7.ControlNodes".cmSepaGripperAxisC.commands.selectSetPosition := 4; END_IF;
   "Unit1.Em7.ControlNodes".cm.Command.sepaGripperAxisC.posAbsolute[4] := #_w1;
END_REGION

REGION Network 158: CmSepaGripperAxisC Position Absolute Position5
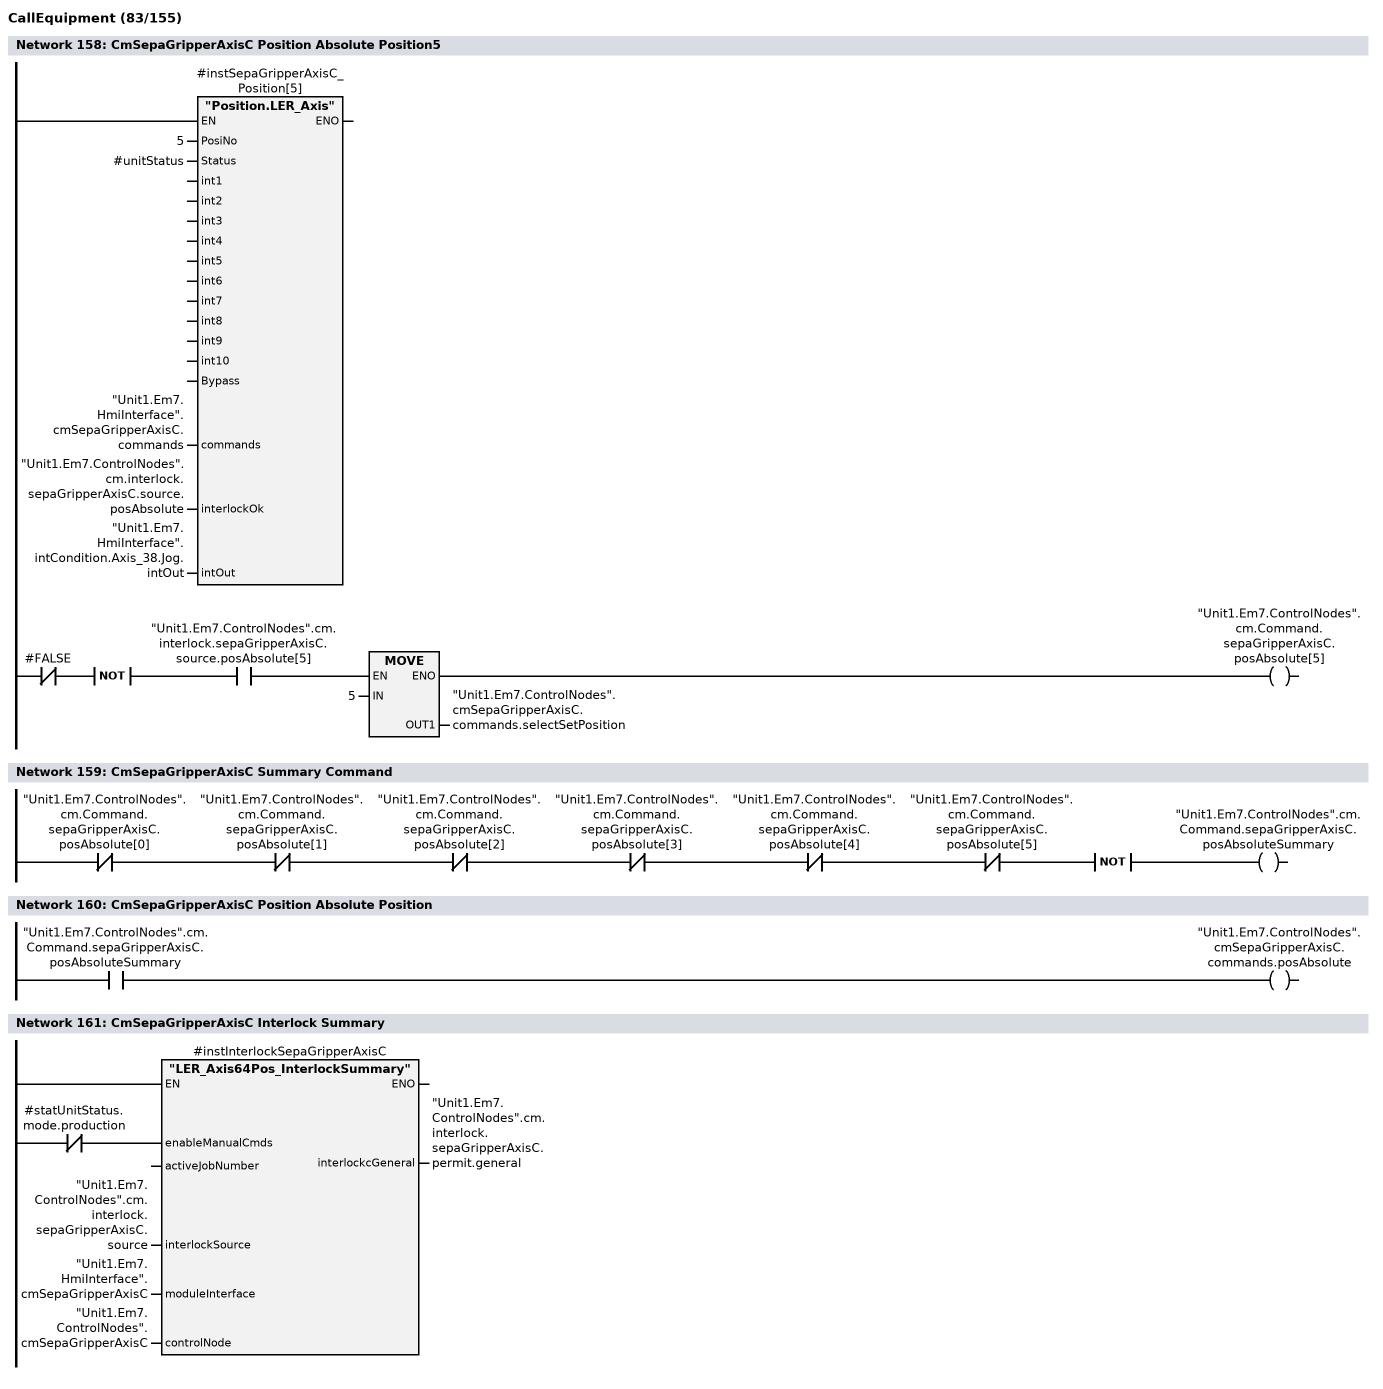
   RUNG wire#powerrail
      #instSepaGripperAxisC_Position[5](PosiNo := 5, Status := #unitStatus, int1 :=, int2 :=, int3 :=, int4 :=, int5 :=, int6 :=, int7 :=, int8 :=, int9 :=, int10 :=, Bypass :=, commands := "Unit1.Em7.HmiInterface".cmSepaGripperAxisC.commands, interlockOk := "Unit1.Em7.ControlNodes".cm.interlock.sepaGripperAxisC.source.posAbsolute, intOut := "Unit1.Em7.HmiInterface".intCondition.Axis_38.Jog.intOut)
   END_RUNG
   RUNG wire#powerrail
      I_Contact( #FALSE )
      Not()
      Contact( "Unit1.Em7.ControlNodes".cm.interlock.sepaGripperAxisC.source.posAbsolute[5] )
      Move(in := 5, out1 => "Unit1.Em7.ControlNodes".cmSepaGripperAxisC.commands.selectSetPosition)
      Coil( "Unit1.Em7.ControlNodes".cm.Command.sepaGripperAxisC.posAbsolute[5] )
   END_RUNG
   // the same network as SCL:
   #instSepaGripperAxisC_Position[5](PosiNo := 5,   // "Position.LER_Axis"
                           Status := #unitStatus,
                           commands := "Unit1.Em7.HmiInterface".cmSepaGripperAxisC.commands,
                           interlockOk := "Unit1.Em7.ControlNodes".cm.interlock.sepaGripperAxisC.source.posAbsolute,
                           intOut := "Unit1.Em7.HmiInterface".intCondition.Axis_38.Jog.intOut);
   #_w1 := NOT (NOT #FALSE) AND "Unit1.Em7.ControlNodes".cm.interlock.sepaGripperAxisC.source.posAbsolute[5];
   IF #_w1 THEN "Unit1.Em7.ControlNodes".cmSepaGripperAxisC.commands.selectSetPosition := 5; END_IF;
   "Unit1.Em7.ControlNodes".cm.Command.sepaGripperAxisC.posAbsolute[5] := #_w1;
END_REGION

REGION Network 159: CmSepaGripperAxisC Summary Command
   RUNG wire#powerrail
      I_Contact( "Unit1.Em7.ControlNodes".cm.Command.sepaGripperAxisC.posAbsolute[0] )
      I_Contact( "Unit1.Em7.ControlNodes".cm.Command.sepaGripperAxisC.posAbsolute[1] )
      I_Contact( "Unit1.Em7.ControlNodes".cm.Command.sepaGripperAxisC.posAbsolute[2] )
      I_Contact( "Unit1.Em7.ControlNodes".cm.Command.sepaGripperAxisC.posAbsolute[3] )
      I_Contact( "Unit1.Em7.ControlNodes".cm.Command.sepaGripperAxisC.posAbsolute[4] )
      I_Contact( "Unit1.Em7.ControlNodes".cm.Command.sepaGripperAxisC.posAbsolute[5] )
      Not()
      Coil( "Unit1.Em7.ControlNodes".cm.Command.sepaGripperAxisC.posAbsoluteSummary )
   END_RUNG
   // the same network as SCL:
   "Unit1.Em7.ControlNodes".cm.Command.sepaGripperAxisC.posAbsoluteSummary := NOT (NOT "Unit1.Em7.ControlNodes".cm.Command.sepaGripperAxisC.posAbsolute[0] AND NOT "Unit1.Em7.ControlNodes".cm.Command.sepaGripperAxisC.posAbsolute[1] AND NOT "Unit1.Em7.ControlNodes".cm.Command.sepaGripperAxisC.posAbsolute[2] AND NOT "Unit1.Em7.ControlNodes".cm.Command.sepaGripperAxisC.posAbsolute[3] AND NOT "Unit1.Em7.ControlNodes".cm.Command.sepaGripperAxisC.posAbsolute[4] AND NOT "Unit1.Em7.ControlNodes".cm.Command.sepaGripperAxisC.posAbsolute[5]);
END_REGION

REGION Network 160: CmSepaGripperAxisC Position Absolute Position
   RUNG wire#powerrail
      Contact( "Unit1.Em7.ControlNodes".cm.Command.sepaGripperAxisC.posAbsoluteSummary )
      Coil( "Unit1.Em7.ControlNodes".cmSepaGripperAxisC.commands.posAbsolute )
   END_RUNG
   // the same network as SCL:
   "Unit1.Em7.ControlNodes".cmSepaGripperAxisC.commands.posAbsolute := "Unit1.Em7.ControlNodes".cm.Command.sepaGripperAxisC.posAbsoluteSummary;
END_REGION

REGION Network 161: CmSepaGripperAxisC Interlock Summary
   RUNG wire#powerrail
      #instInterlockSepaGripperAxisC(enableManualCmds := wire#w1, activeJobNumber :=, interlockSource := "Unit1.Em7.ControlNodes".cm.interlock.sepaGripperAxisC.source, moduleInterface := "Unit1.Em7.HmiInterface".cmSepaGripperAxisC, controlNode := "Unit1.Em7.ControlNodes".cmSepaGripperAxisC, interlockcGeneral => "Unit1.Em7.ControlNodes".cm.interlock.sepaGripperAxisC.permit.general)
   END_RUNG
   RUNG wire#powerrail
      I_Contact( #statUnitStatus.mode.production )
   END_RUNG wire#w1
   // the same network as SCL:
   #instInterlockSepaGripperAxisC(enableManualCmds := NOT #statUnitStatus.mode.production,   // "LER_Axis64Pos_InterlockSummary"
                           interlockSource := "Unit1.Em7.ControlNodes".cm.interlock.sepaGripperAxisC.source,
                           moduleInterface := "Unit1.Em7.HmiInterface".cmSepaGripperAxisC,
                           controlNode := "Unit1.Em7.ControlNodes".cmSepaGripperAxisC,
                           interlockcGeneral => "Unit1.Em7.ControlNodes".cm.interlock.sepaGripperAxisC.permit.general);
END_REGION

REGION Network 162: CmSepaGripperAxisC velocity/speed
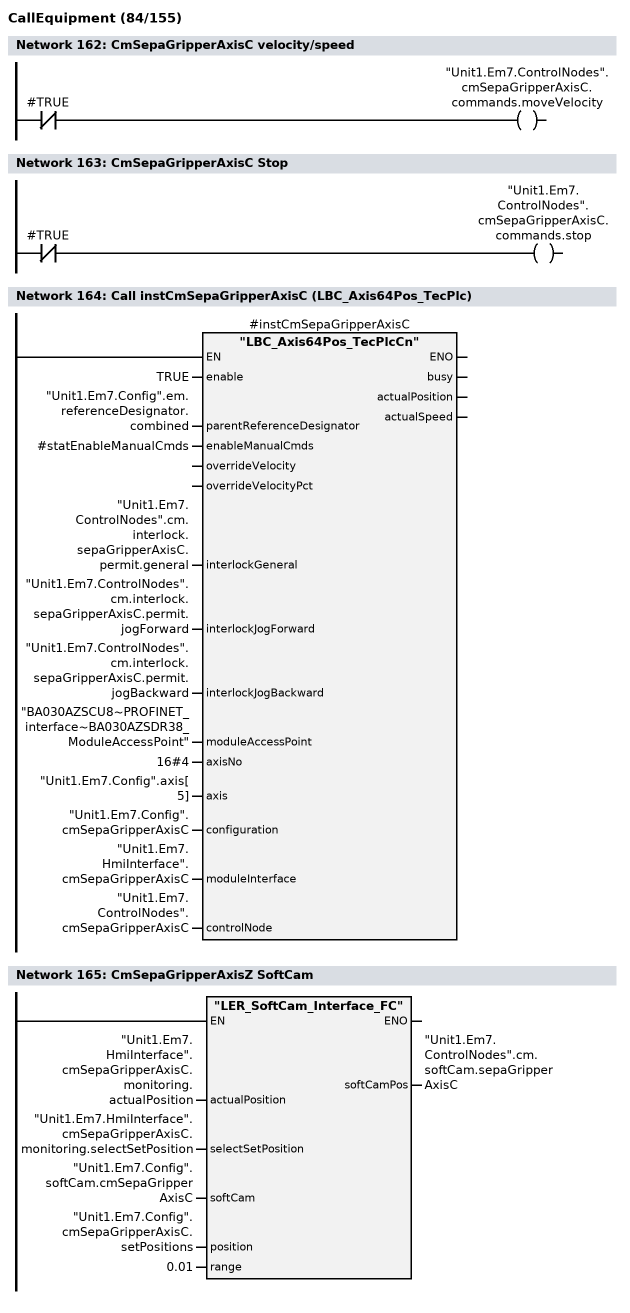
   RUNG wire#powerrail
      I_Contact( #TRUE )
      Coil( "Unit1.Em7.ControlNodes".cmSepaGripperAxisC.commands.moveVelocity )
   END_RUNG
   // the same network as SCL:
   "Unit1.Em7.ControlNodes".cmSepaGripperAxisC.commands.moveVelocity := NOT #TRUE;
END_REGION

REGION Network 163: CmSepaGripperAxisC Stop
   RUNG wire#powerrail
      I_Contact( #TRUE )
      Coil( "Unit1.Em7.ControlNodes".cmSepaGripperAxisC.commands.stop )
   END_RUNG
   // the same network as SCL:
   "Unit1.Em7.ControlNodes".cmSepaGripperAxisC.commands.stop := NOT #TRUE;
END_REGION

REGION Network 164: Call instCmSepaGripperAxisC (LBC_Axis64Pos_TecPlc)
   RUNG wire#powerrail
      #instCmSepaGripperAxisC(enable := TRUE, parentReferenceDesignator := "Unit1.Em7.Config".em.referenceDesignator.combined, enableManualCmds := #statEnableManualCmds, overrideVelocity :=, overrideVelocityPct :=, interlockGeneral := "Unit1.Em7.ControlNodes".cm.interlock.sepaGripperAxisC.permit.general, interlockJogForward := "Unit1.Em7.ControlNodes".cm.interlock.sepaGripperAxisC.permit.jogForward, interlockJogBackward := "Unit1.Em7.ControlNodes".cm.interlock.sepaGripperAxisC.permit.jogBackward, moduleAccessPoint := "BA030AZSCU8~PROFINET_interface~BA030AZSDR38_ModuleAccessPoint", axisNo := 16#4, axis := "Unit1.Em7.Config".axis[5], configuration := "Unit1.Em7.Config".cmSepaGripperAxisC, moduleInterface := "Unit1.Em7.HmiInterface".cmSepaGripperAxisC, controlNode := "Unit1.Em7.ControlNodes".cmSepaGripperAxisC, busy =>, actualPosition =>, actualSpeed =>)
   END_RUNG
   // the same network as SCL:
   #instCmSepaGripperAxisC(enable := TRUE,   // "LBC_Axis64Pos_TecPlcCn"
                           parentReferenceDesignator := "Unit1.Em7.Config".em.referenceDesignator.combined,
                           enableManualCmds := #statEnableManualCmds,
                           interlockGeneral := "Unit1.Em7.ControlNodes".cm.interlock.sepaGripperAxisC.permit.general,
                           interlockJogForward := "Unit1.Em7.ControlNodes".cm.interlock.sepaGripperAxisC.permit.jogForward,
                           interlockJogBackward := "Unit1.Em7.ControlNodes".cm.interlock.sepaGripperAxisC.permit.jogBackward,
                           moduleAccessPoint := "BA030AZSCU8~PROFINET_interface~BA030AZSDR38_ModuleAccessPoint",
                           axisNo := 16#4,
                           axis := "Unit1.Em7.Config".axis[5],
                           configuration := "Unit1.Em7.Config".cmSepaGripperAxisC,
                           moduleInterface := "Unit1.Em7.HmiInterface".cmSepaGripperAxisC,
                           controlNode := "Unit1.Em7.ControlNodes".cmSepaGripperAxisC);
END_REGION

REGION Network 165: CmSepaGripperAxisZ SoftCam
   RUNG wire#powerrail
      "LER_SoftCam_Interface_FC"(actualPosition := "Unit1.Em7.HmiInterface".cmSepaGripperAxisC.monitoring.actualPosition, selectSetPosition := "Unit1.Em7.HmiInterface".cmSepaGripperAxisC.monitoring.selectSetPosition, softCam := "Unit1.Em7.Config".softCam.cmSepaGripperAxisC, position := "Unit1.Em7.Config".cmSepaGripperAxisC.setPositions, range := 0.01, softCamPos => "Unit1.Em7.ControlNodes".cm.softCam.sepaGripperAxisC)
   END_RUNG
   // the same network as SCL:
   "LER_SoftCam_Interface_FC"(actualPosition := "Unit1.Em7.HmiInterface".cmSepaGripperAxisC.monitoring.actualPosition,
                           selectSetPosition := "Unit1.Em7.HmiInterface".cmSepaGripperAxisC.monitoring.selectSetPosition,
                           softCam := "Unit1.Em7.Config".softCam.cmSepaGripperAxisC,
                           position := "Unit1.Em7.Config".cmSepaGripperAxisC.setPositions,
                           range := 0.01,
                           softCamPos => "Unit1.Em7.ControlNodes".cm.softCam.sepaGripperAxisC);
END_REGION

REGION Network 167: JRWinderRearAxisY Enable
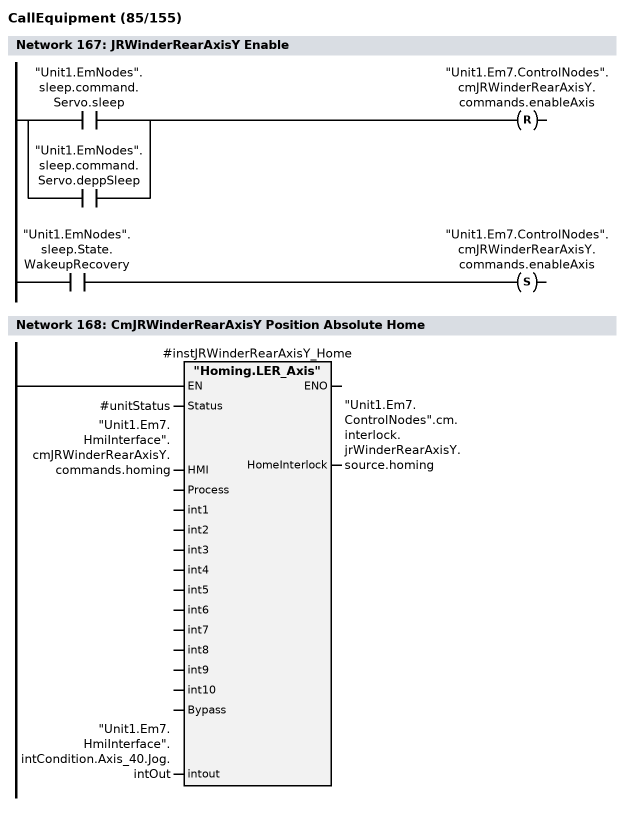
   RUNG wire#powerrail
      Contact( "Unit1.EmNodes".sleep.command.Servo.sleep )
      wire#w1
      R_Coil( "Unit1.Em7.ControlNodes".cmJRWinderRearAxisY.commands.enableAxis )
   END_RUNG
   RUNG wire#powerrail
      Contact( "Unit1.EmNodes".sleep.command.Servo.deppSleep )
   END_RUNG wire#w1
   RUNG wire#powerrail
      Contact( "Unit1.EmNodes".sleep.State.WakeupRecovery )
      S_Coil( "Unit1.Em7.ControlNodes".cmJRWinderRearAxisY.commands.enableAxis )
   END_RUNG
   // the same network as SCL:
   IF "Unit1.EmNodes".sleep.command.Servo.sleep OR "Unit1.EmNodes".sleep.command.Servo.deppSleep THEN
       "Unit1.Em7.ControlNodes".cmJRWinderRearAxisY.commands.enableAxis := FALSE;
   END_IF;
   IF "Unit1.EmNodes".sleep.State.WakeupRecovery THEN
       "Unit1.Em7.ControlNodes".cmJRWinderRearAxisY.commands.enableAxis := TRUE;
   END_IF;
END_REGION

REGION Network 168: CmJRWinderRearAxisY Position Absolute Home
   RUNG wire#powerrail
      #instJRWinderRearAxisY_Home(Status := #unitStatus, HMI := "Unit1.Em7.HmiInterface".cmJRWinderRearAxisY.commands.homing, Process :=, int1 :=, int2 :=, int3 :=, int4 :=, int5 :=, int6 :=, int7 :=, int8 :=, int9 :=, int10 :=, Bypass :=, intout := "Unit1.Em7.HmiInterface".intCondition.Axis_40.Jog.intOut, HomeInterlock => "Unit1.Em7.ControlNodes".cm.interlock.jrWinderRearAxisY.source.homing)
   END_RUNG
   // the same network as SCL:
   #instJRWinderRearAxisY_Home(Status := #unitStatus,   // "Homing.LER_Axis"
                           HMI := "Unit1.Em7.HmiInterface".cmJRWinderRearAxisY.commands.homing,
                           intout := "Unit1.Em7.HmiInterface".intCondition.Axis_40.Jog.intOut,
                           HomeInterlock => "Unit1.Em7.ControlNodes".cm.interlock.jrWinderRearAxisY.source.homing);
END_REGION

REGION Network 169: CmJRWinderRearAxisY Position Absolute Jog
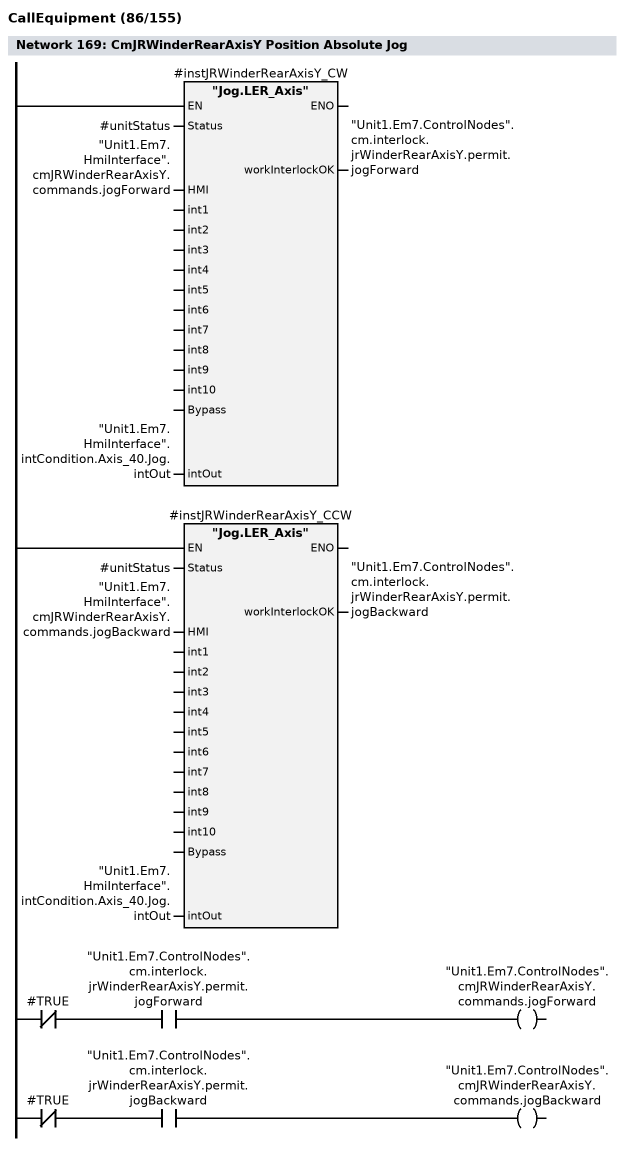
   RUNG wire#powerrail
      #instJRWinderRearAxisY_CW(Status := #unitStatus, HMI := "Unit1.Em7.HmiInterface".cmJRWinderRearAxisY.commands.jogForward, int1 :=, int2 :=, int3 :=, int4 :=, int5 :=, int6 :=, int7 :=, int8 :=, int9 :=, int10 :=, Bypass :=, intOut := "Unit1.Em7.HmiInterface".intCondition.Axis_40.Jog.intOut, workInterlockOK => "Unit1.Em7.ControlNodes".cm.interlock.jrWinderRearAxisY.permit.jogForward)
   END_RUNG
   RUNG wire#powerrail
      #instJRWinderRearAxisY_CCW(Status := #unitStatus, HMI := "Unit1.Em7.HmiInterface".cmJRWinderRearAxisY.commands.jogBackward, int1 :=, int2 :=, int3 :=, int4 :=, int5 :=, int6 :=, int7 :=, int8 :=, int9 :=, int10 :=, Bypass :=, intOut := "Unit1.Em7.HmiInterface".intCondition.Axis_40.Jog.intOut, workInterlockOK => "Unit1.Em7.ControlNodes".cm.interlock.jrWinderRearAxisY.permit.jogBackward)
   END_RUNG
   RUNG wire#powerrail
      I_Contact( #TRUE )
      Contact( "Unit1.Em7.ControlNodes".cm.interlock.jrWinderRearAxisY.permit.jogForward )
      Coil( "Unit1.Em7.ControlNodes".cmJRWinderRearAxisY.commands.jogForward )
   END_RUNG
   RUNG wire#powerrail
      I_Contact( #TRUE )
      Contact( "Unit1.Em7.ControlNodes".cm.interlock.jrWinderRearAxisY.permit.jogBackward )
      Coil( "Unit1.Em7.ControlNodes".cmJRWinderRearAxisY.commands.jogBackward )
   END_RUNG
   // the same network as SCL:
   #instJRWinderRearAxisY_CW(Status := #unitStatus,   // "Jog.LER_Axis"
                           HMI := "Unit1.Em7.HmiInterface".cmJRWinderRearAxisY.commands.jogForward,
                           intOut := "Unit1.Em7.HmiInterface".intCondition.Axis_40.Jog.intOut,
                           workInterlockOK => "Unit1.Em7.ControlNodes".cm.interlock.jrWinderRearAxisY.permit.jogForward);
   #instJRWinderRearAxisY_CCW(Status := #unitStatus,   // "Jog.LER_Axis"
                           HMI := "Unit1.Em7.HmiInterface".cmJRWinderRearAxisY.commands.jogBackward,
                           intOut := "Unit1.Em7.HmiInterface".intCondition.Axis_40.Jog.intOut,
                           workInterlockOK => "Unit1.Em7.ControlNodes".cm.interlock.jrWinderRearAxisY.permit.jogBackward);
   "Unit1.Em7.ControlNodes".cmJRWinderRearAxisY.commands.jogForward := NOT #TRUE AND "Unit1.Em7.ControlNodes".cm.interlock.jrWinderRearAxisY.permit.jogForward;
   "Unit1.Em7.ControlNodes".cmJRWinderRearAxisY.commands.jogBackward := NOT #TRUE AND "Unit1.Em7.ControlNodes".cm.interlock.jrWinderRearAxisY.permit.jogBackward;
END_REGION

REGION Network 170: CmJRWinderRearAxisY Position Absolute Position0
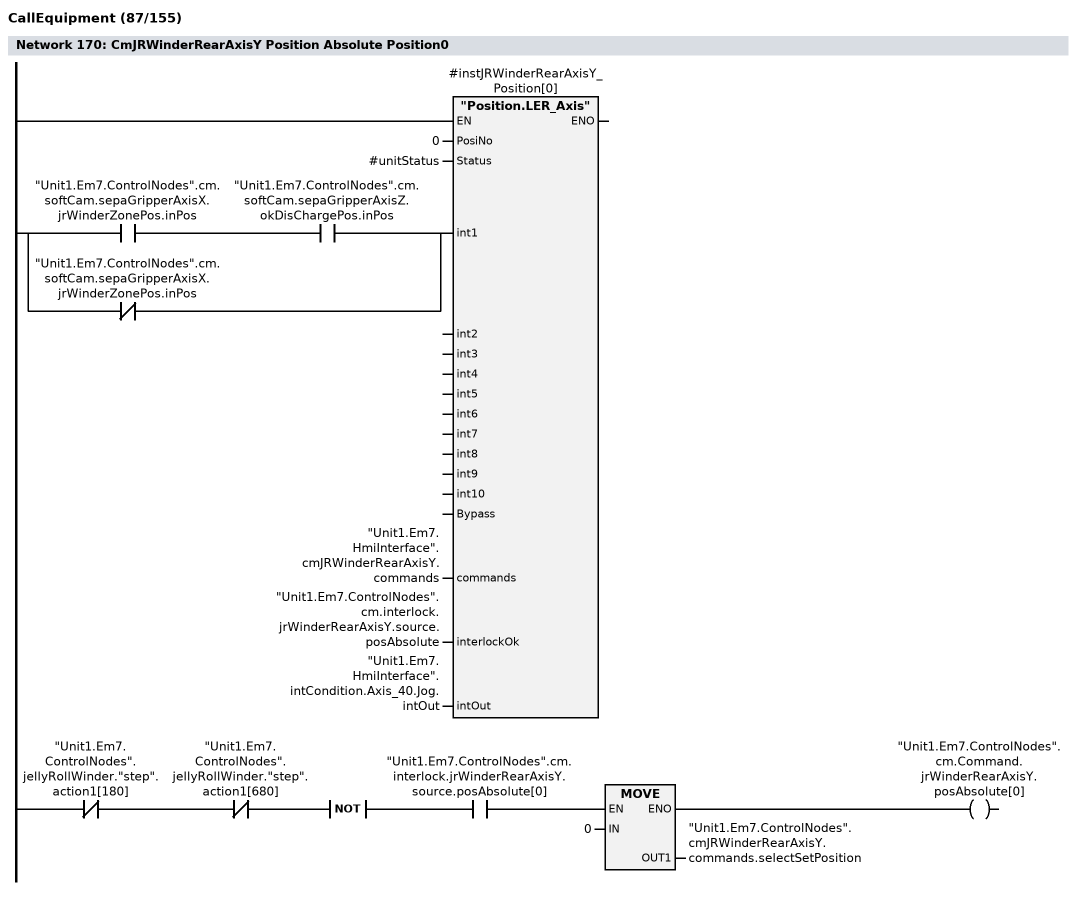
   RUNG wire#powerrail
      #instJRWinderRearAxisY_Position[0](int1 := wire#w1, PosiNo := 0, Status := #unitStatus, int2 :=, int3 :=, int4 :=, int5 :=, int6 :=, int7 :=, int8 :=, int9 :=, int10 :=, Bypass :=, commands := "Unit1.Em7.HmiInterface".cmJRWinderRearAxisY.commands, interlockOk := "Unit1.Em7.ControlNodes".cm.interlock.jrWinderRearAxisY.source.posAbsolute, intOut := "Unit1.Em7.HmiInterface".intCondition.Axis_40.Jog.intOut)
   END_RUNG
   RUNG wire#powerrail
      Contact( "Unit1.Em7.ControlNodes".cm.softCam.sepaGripperAxisX.jrWinderZonePos.inPos )
      Contact( "Unit1.Em7.ControlNodes".cm.softCam.sepaGripperAxisZ.okDisChargePos.inPos )
   END_RUNG wire#w1
   RUNG wire#powerrail
      I_Contact( "Unit1.Em7.ControlNodes".cm.softCam.sepaGripperAxisX.jrWinderZonePos.inPos )
   END_RUNG wire#w1
   RUNG wire#powerrail
      I_Contact( "Unit1.Em7.ControlNodes".jellyRollWinder."step".action1[180] )
      I_Contact( "Unit1.Em7.ControlNodes".jellyRollWinder."step".action1[680] )
      Not()
      Contact( "Unit1.Em7.ControlNodes".cm.interlock.jrWinderRearAxisY.source.posAbsolute[0] )
      Move(in := 0, out1 => "Unit1.Em7.ControlNodes".cmJRWinderRearAxisY.commands.selectSetPosition)
      Coil( "Unit1.Em7.ControlNodes".cm.Command.jrWinderRearAxisY.posAbsolute[0] )
   END_RUNG
   // the same network as SCL:
   #instJRWinderRearAxisY_Position[0](PosiNo := 0,   // "Position.LER_Axis"
                           Status := #unitStatus,
                           int1 := ("Unit1.Em7.ControlNodes".cm.softCam.sepaGripperAxisX.jrWinderZonePos.inPos AND "Unit1.Em7.ControlNodes".cm.softCam.sepaGripperAxisZ.okDisChargePos.inPos) OR NOT "Unit1.Em7.ControlNodes".cm.softCam.sepaGripperAxisX.jrWinderZonePos.inPos,
                           commands := "Unit1.Em7.HmiInterface".cmJRWinderRearAxisY.commands,
                           interlockOk := "Unit1.Em7.ControlNodes".cm.interlock.jrWinderRearAxisY.source.posAbsolute,
                           intOut := "Unit1.Em7.HmiInterface".intCondition.Axis_40.Jog.intOut);
   #_w1 := NOT (NOT "Unit1.Em7.ControlNodes".jellyRollWinder."step".action1[180] AND NOT "Unit1.Em7.ControlNodes".jellyRollWinder."step".action1[680]) AND "Unit1.Em7.ControlNodes".cm.interlock.jrWinderRearAxisY.source.posAbsolute[0];
   IF #_w1 THEN "Unit1.Em7.ControlNodes".cmJRWinderRearAxisY.commands.selectSetPosition := 0; END_IF;
   "Unit1.Em7.ControlNodes".cm.Command.jrWinderRearAxisY.posAbsolute[0] := #_w1;
END_REGION

REGION Network 171: CmJRWinderRearAxisY Position Absolute Position1
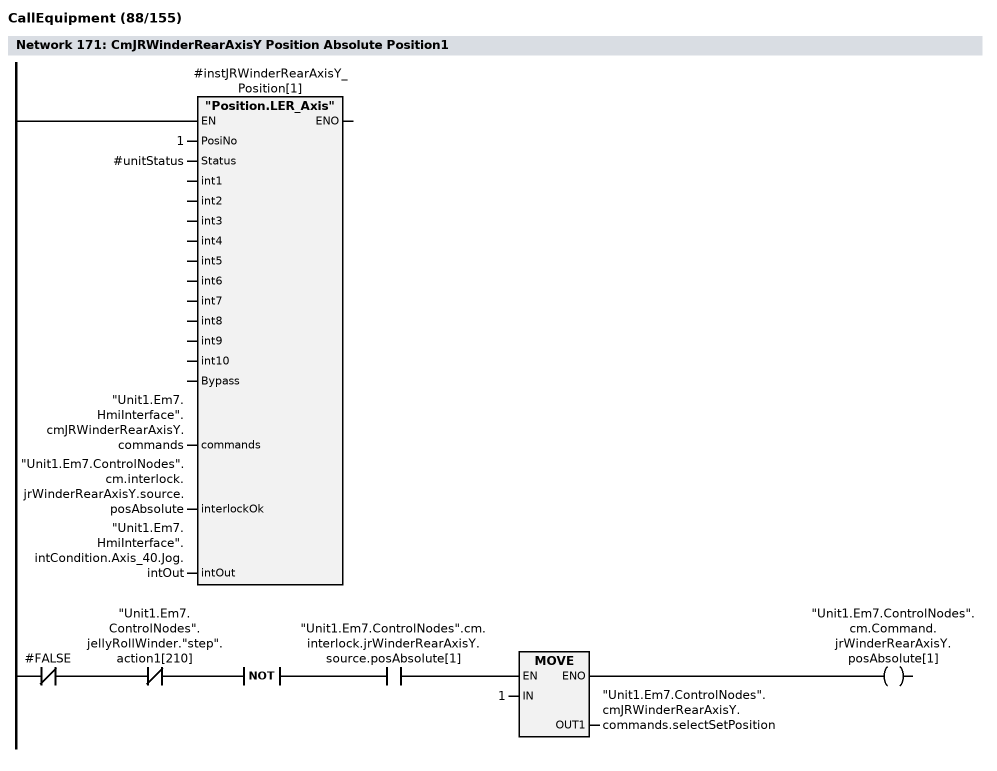
   RUNG wire#powerrail
      #instJRWinderRearAxisY_Position[1](PosiNo := 1, Status := #unitStatus, int1 :=, int2 :=, int3 :=, int4 :=, int5 :=, int6 :=, int7 :=, int8 :=, int9 :=, int10 :=, Bypass :=, commands := "Unit1.Em7.HmiInterface".cmJRWinderRearAxisY.commands, interlockOk := "Unit1.Em7.ControlNodes".cm.interlock.jrWinderRearAxisY.source.posAbsolute, intOut := "Unit1.Em7.HmiInterface".intCondition.Axis_40.Jog.intOut)
   END_RUNG
   RUNG wire#powerrail
      I_Contact( #FALSE )
      I_Contact( "Unit1.Em7.ControlNodes".jellyRollWinder."step".action1[210] )
      Not()
      Contact( "Unit1.Em7.ControlNodes".cm.interlock.jrWinderRearAxisY.source.posAbsolute[1] )
      Move(in := 1, out1 => "Unit1.Em7.ControlNodes".cmJRWinderRearAxisY.commands.selectSetPosition)
      Coil( "Unit1.Em7.ControlNodes".cm.Command.jrWinderRearAxisY.posAbsolute[1] )
   END_RUNG
   // the same network as SCL:
   #instJRWinderRearAxisY_Position[1](PosiNo := 1,   // "Position.LER_Axis"
                           Status := #unitStatus,
                           commands := "Unit1.Em7.HmiInterface".cmJRWinderRearAxisY.commands,
                           interlockOk := "Unit1.Em7.ControlNodes".cm.interlock.jrWinderRearAxisY.source.posAbsolute,
                           intOut := "Unit1.Em7.HmiInterface".intCondition.Axis_40.Jog.intOut);
   #_w1 := NOT (NOT #FALSE AND NOT "Unit1.Em7.ControlNodes".jellyRollWinder."step".action1[210]) AND "Unit1.Em7.ControlNodes".cm.interlock.jrWinderRearAxisY.source.posAbsolute[1];
   IF #_w1 THEN "Unit1.Em7.ControlNodes".cmJRWinderRearAxisY.commands.selectSetPosition := 1; END_IF;
   "Unit1.Em7.ControlNodes".cm.Command.jrWinderRearAxisY.posAbsolute[1] := #_w1;
END_REGION

REGION Network 172: CmJRWinderRearAxisY Position Absolute Position2
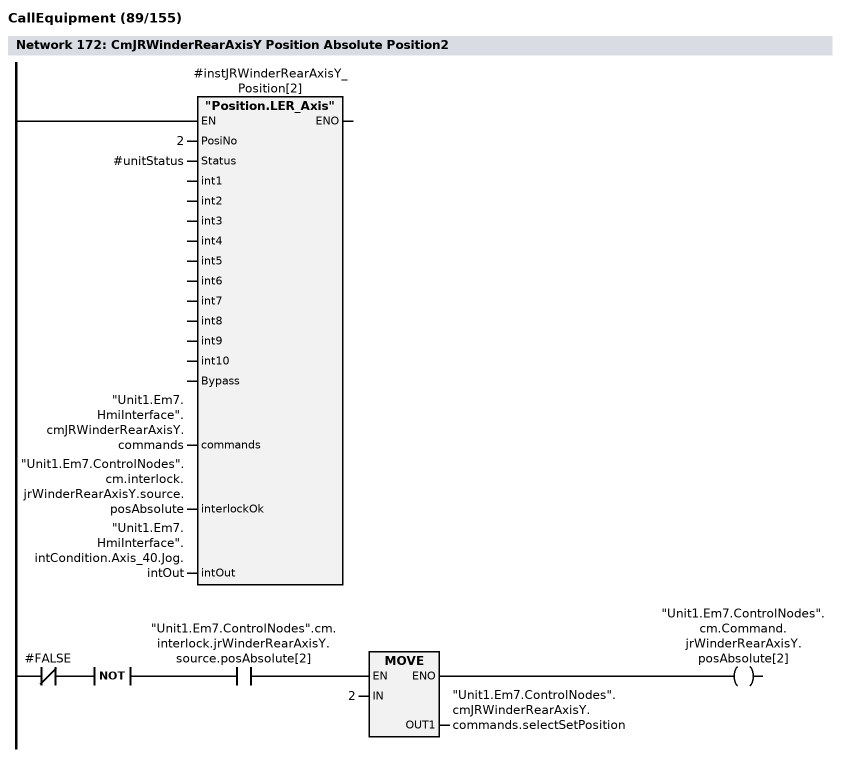
   RUNG wire#powerrail
      #instJRWinderRearAxisY_Position[2](PosiNo := 2, Status := #unitStatus, int1 :=, int2 :=, int3 :=, int4 :=, int5 :=, int6 :=, int7 :=, int8 :=, int9 :=, int10 :=, Bypass :=, commands := "Unit1.Em7.HmiInterface".cmJRWinderRearAxisY.commands, interlockOk := "Unit1.Em7.ControlNodes".cm.interlock.jrWinderRearAxisY.source.posAbsolute, intOut := "Unit1.Em7.HmiInterface".intCondition.Axis_40.Jog.intOut)
   END_RUNG
   RUNG wire#powerrail
      I_Contact( #FALSE )
      Not()
      Contact( "Unit1.Em7.ControlNodes".cm.interlock.jrWinderRearAxisY.source.posAbsolute[2] )
      Move(in := 2, out1 => "Unit1.Em7.ControlNodes".cmJRWinderRearAxisY.commands.selectSetPosition)
      Coil( "Unit1.Em7.ControlNodes".cm.Command.jrWinderRearAxisY.posAbsolute[2] )
   END_RUNG
   // the same network as SCL:
   #instJRWinderRearAxisY_Position[2](PosiNo := 2,   // "Position.LER_Axis"
                           Status := #unitStatus,
                           commands := "Unit1.Em7.HmiInterface".cmJRWinderRearAxisY.commands,
                           interlockOk := "Unit1.Em7.ControlNodes".cm.interlock.jrWinderRearAxisY.source.posAbsolute,
                           intOut := "Unit1.Em7.HmiInterface".intCondition.Axis_40.Jog.intOut);
   #_w1 := NOT (NOT #FALSE) AND "Unit1.Em7.ControlNodes".cm.interlock.jrWinderRearAxisY.source.posAbsolute[2];
   IF #_w1 THEN "Unit1.Em7.ControlNodes".cmJRWinderRearAxisY.commands.selectSetPosition := 2; END_IF;
   "Unit1.Em7.ControlNodes".cm.Command.jrWinderRearAxisY.posAbsolute[2] := #_w1;
END_REGION

REGION Network 173: CmJRWinderRearAxisY Position Absolute Position3
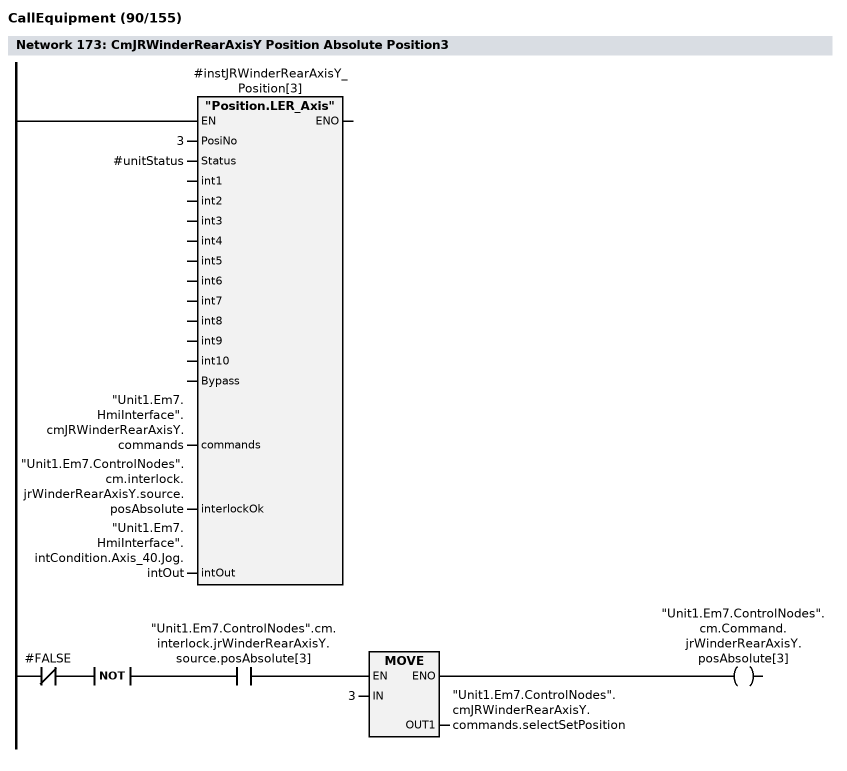
   RUNG wire#powerrail
      #instJRWinderRearAxisY_Position[3](PosiNo := 3, Status := #unitStatus, int1 :=, int2 :=, int3 :=, int4 :=, int5 :=, int6 :=, int7 :=, int8 :=, int9 :=, int10 :=, Bypass :=, commands := "Unit1.Em7.HmiInterface".cmJRWinderRearAxisY.commands, interlockOk := "Unit1.Em7.ControlNodes".cm.interlock.jrWinderRearAxisY.source.posAbsolute, intOut := "Unit1.Em7.HmiInterface".intCondition.Axis_40.Jog.intOut)
   END_RUNG
   RUNG wire#powerrail
      I_Contact( #FALSE )
      Not()
      Contact( "Unit1.Em7.ControlNodes".cm.interlock.jrWinderRearAxisY.source.posAbsolute[3] )
      Move(in := 3, out1 => "Unit1.Em7.ControlNodes".cmJRWinderRearAxisY.commands.selectSetPosition)
      Coil( "Unit1.Em7.ControlNodes".cm.Command.jrWinderRearAxisY.posAbsolute[3] )
   END_RUNG
   // the same network as SCL:
   #instJRWinderRearAxisY_Position[3](PosiNo := 3,   // "Position.LER_Axis"
                           Status := #unitStatus,
                           commands := "Unit1.Em7.HmiInterface".cmJRWinderRearAxisY.commands,
                           interlockOk := "Unit1.Em7.ControlNodes".cm.interlock.jrWinderRearAxisY.source.posAbsolute,
                           intOut := "Unit1.Em7.HmiInterface".intCondition.Axis_40.Jog.intOut);
   #_w1 := NOT (NOT #FALSE) AND "Unit1.Em7.ControlNodes".cm.interlock.jrWinderRearAxisY.source.posAbsolute[3];
   IF #_w1 THEN "Unit1.Em7.ControlNodes".cmJRWinderRearAxisY.commands.selectSetPosition := 3; END_IF;
   "Unit1.Em7.ControlNodes".cm.Command.jrWinderRearAxisY.posAbsolute[3] := #_w1;
END_REGION

REGION Network 174: CmJRWinderRearAxisY Position Absolute Position4
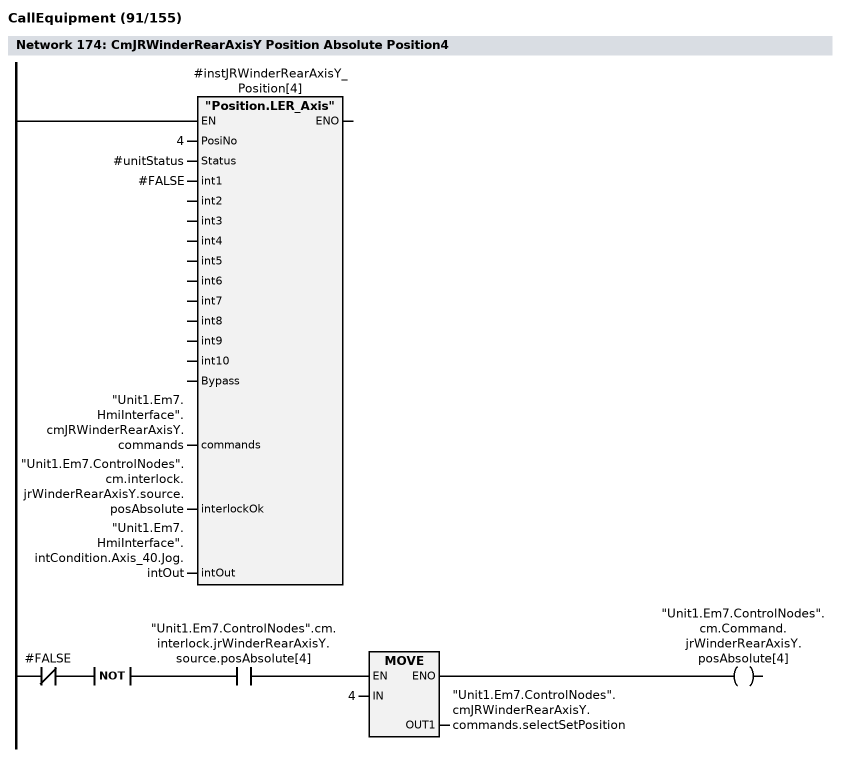
   RUNG wire#powerrail
      #instJRWinderRearAxisY_Position[4](PosiNo := 4, Status := #unitStatus, int1 := #FALSE, int2 :=, int3 :=, int4 :=, int5 :=, int6 :=, int7 :=, int8 :=, int9 :=, int10 :=, Bypass :=, commands := "Unit1.Em7.HmiInterface".cmJRWinderRearAxisY.commands, interlockOk := "Unit1.Em7.ControlNodes".cm.interlock.jrWinderRearAxisY.source.posAbsolute, intOut := "Unit1.Em7.HmiInterface".intCondition.Axis_40.Jog.intOut)
   END_RUNG
   RUNG wire#powerrail
      I_Contact( #FALSE )
      Not()
      Contact( "Unit1.Em7.ControlNodes".cm.interlock.jrWinderRearAxisY.source.posAbsolute[4] )
      Move(in := 4, out1 => "Unit1.Em7.ControlNodes".cmJRWinderRearAxisY.commands.selectSetPosition)
      Coil( "Unit1.Em7.ControlNodes".cm.Command.jrWinderRearAxisY.posAbsolute[4] )
   END_RUNG
   // the same network as SCL:
   #instJRWinderRearAxisY_Position[4](PosiNo := 4,   // "Position.LER_Axis"
                           Status := #unitStatus,
                           int1 := #FALSE,
                           commands := "Unit1.Em7.HmiInterface".cmJRWinderRearAxisY.commands,
                           interlockOk := "Unit1.Em7.ControlNodes".cm.interlock.jrWinderRearAxisY.source.posAbsolute,
                           intOut := "Unit1.Em7.HmiInterface".intCondition.Axis_40.Jog.intOut);
   #_w1 := NOT (NOT #FALSE) AND "Unit1.Em7.ControlNodes".cm.interlock.jrWinderRearAxisY.source.posAbsolute[4];
   IF #_w1 THEN "Unit1.Em7.ControlNodes".cmJRWinderRearAxisY.commands.selectSetPosition := 4; END_IF;
   "Unit1.Em7.ControlNodes".cm.Command.jrWinderRearAxisY.posAbsolute[4] := #_w1;
END_REGION

REGION Network 175: CmJRWinderRearAxisY Position Absolute Position5
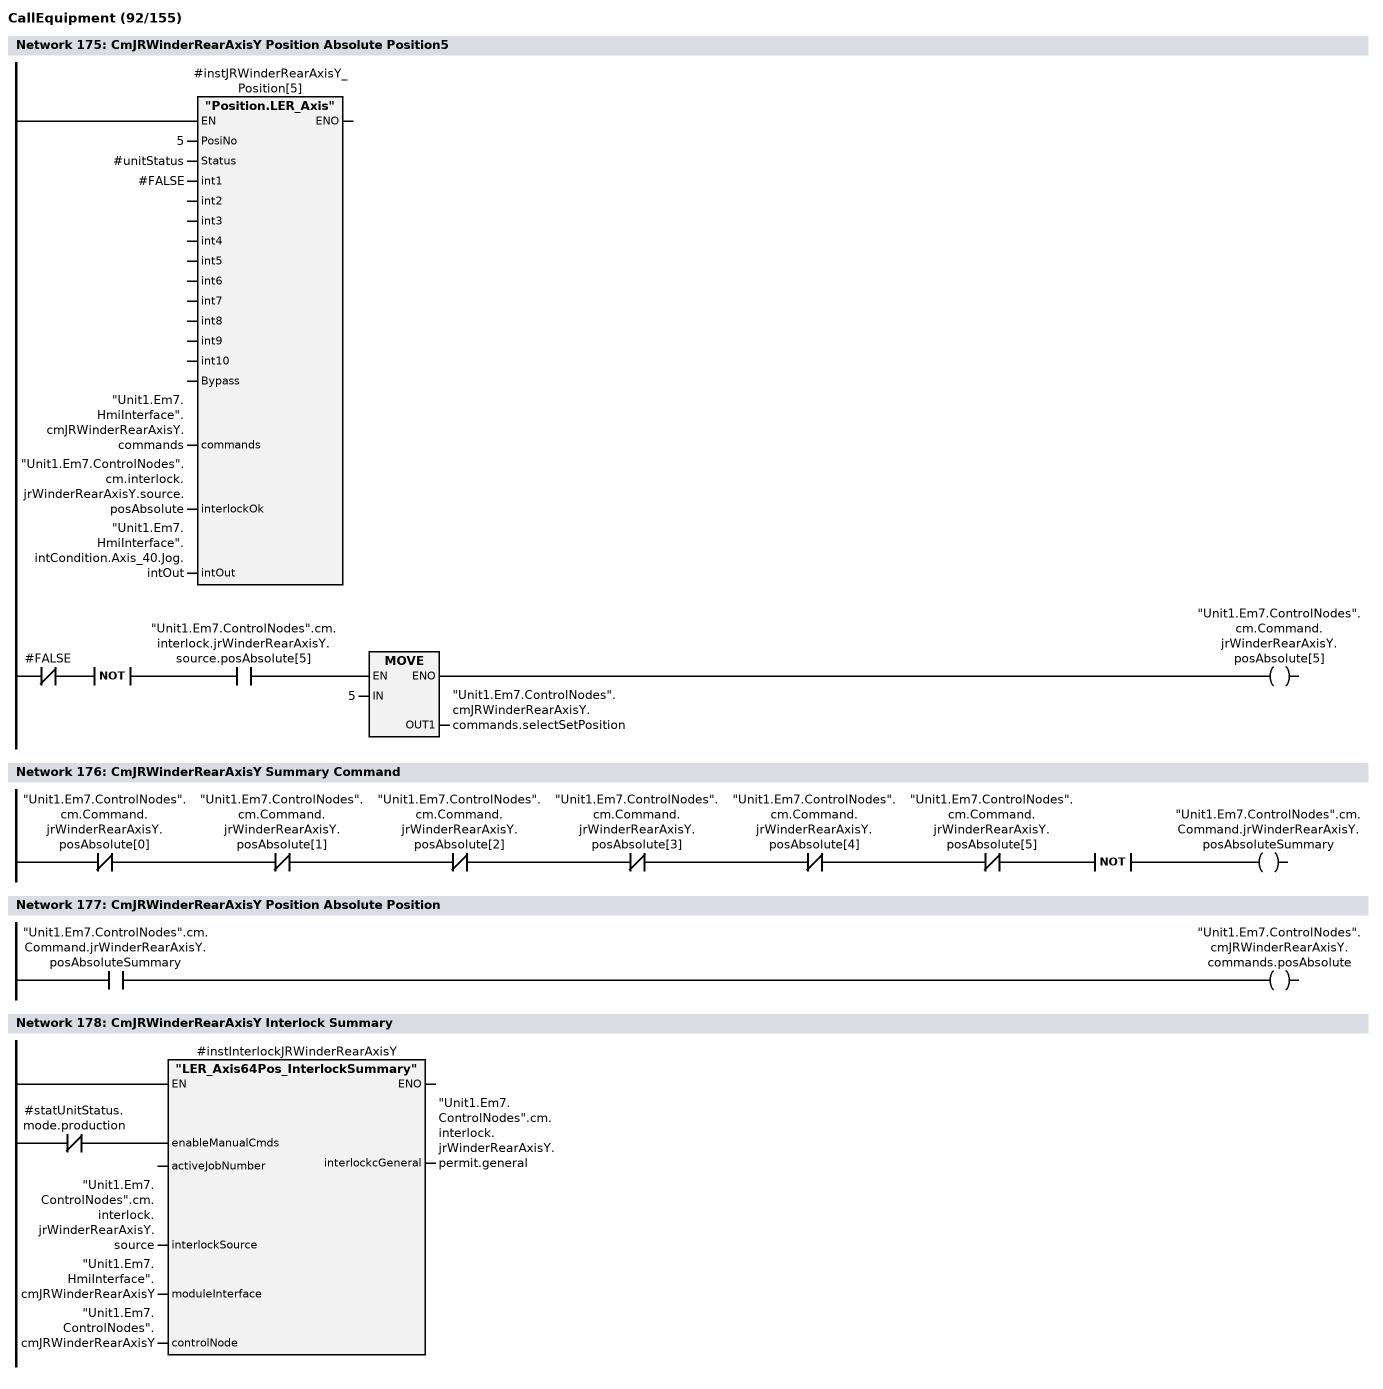
   RUNG wire#powerrail
      #instJRWinderRearAxisY_Position[5](PosiNo := 5, Status := #unitStatus, int1 := #FALSE, int2 :=, int3 :=, int4 :=, int5 :=, int6 :=, int7 :=, int8 :=, int9 :=, int10 :=, Bypass :=, commands := "Unit1.Em7.HmiInterface".cmJRWinderRearAxisY.commands, interlockOk := "Unit1.Em7.ControlNodes".cm.interlock.jrWinderRearAxisY.source.posAbsolute, intOut := "Unit1.Em7.HmiInterface".intCondition.Axis_40.Jog.intOut)
   END_RUNG
   RUNG wire#powerrail
      I_Contact( #FALSE )
      Not()
      Contact( "Unit1.Em7.ControlNodes".cm.interlock.jrWinderRearAxisY.source.posAbsolute[5] )
      Move(in := 5, out1 => "Unit1.Em7.ControlNodes".cmJRWinderRearAxisY.commands.selectSetPosition)
      Coil( "Unit1.Em7.ControlNodes".cm.Command.jrWinderRearAxisY.posAbsolute[5] )
   END_RUNG
   // the same network as SCL:
   #instJRWinderRearAxisY_Position[5](PosiNo := 5,   // "Position.LER_Axis"
                           Status := #unitStatus,
                           int1 := #FALSE,
                           commands := "Unit1.Em7.HmiInterface".cmJRWinderRearAxisY.commands,
                           interlockOk := "Unit1.Em7.ControlNodes".cm.interlock.jrWinderRearAxisY.source.posAbsolute,
                           intOut := "Unit1.Em7.HmiInterface".intCondition.Axis_40.Jog.intOut);
   #_w1 := NOT (NOT #FALSE) AND "Unit1.Em7.ControlNodes".cm.interlock.jrWinderRearAxisY.source.posAbsolute[5];
   IF #_w1 THEN "Unit1.Em7.ControlNodes".cmJRWinderRearAxisY.commands.selectSetPosition := 5; END_IF;
   "Unit1.Em7.ControlNodes".cm.Command.jrWinderRearAxisY.posAbsolute[5] := #_w1;
END_REGION

REGION Network 176: CmJRWinderRearAxisY Summary Command
   RUNG wire#powerrail
      I_Contact( "Unit1.Em7.ControlNodes".cm.Command.jrWinderRearAxisY.posAbsolute[0] )
      I_Contact( "Unit1.Em7.ControlNodes".cm.Command.jrWinderRearAxisY.posAbsolute[1] )
      I_Contact( "Unit1.Em7.ControlNodes".cm.Command.jrWinderRearAxisY.posAbsolute[2] )
      I_Contact( "Unit1.Em7.ControlNodes".cm.Command.jrWinderRearAxisY.posAbsolute[3] )
      I_Contact( "Unit1.Em7.ControlNodes".cm.Command.jrWinderRearAxisY.posAbsolute[4] )
      I_Contact( "Unit1.Em7.ControlNodes".cm.Command.jrWinderRearAxisY.posAbsolute[5] )
      Not()
      Coil( "Unit1.Em7.ControlNodes".cm.Command.jrWinderRearAxisY.posAbsoluteSummary )
   END_RUNG
   // the same network as SCL:
   "Unit1.Em7.ControlNodes".cm.Command.jrWinderRearAxisY.posAbsoluteSummary := NOT (NOT "Unit1.Em7.ControlNodes".cm.Command.jrWinderRearAxisY.posAbsolute[0] AND NOT "Unit1.Em7.ControlNodes".cm.Command.jrWinderRearAxisY.posAbsolute[1] AND NOT "Unit1.Em7.ControlNodes".cm.Command.jrWinderRearAxisY.posAbsolute[2] AND NOT "Unit1.Em7.ControlNodes".cm.Command.jrWinderRearAxisY.posAbsolute[3] AND NOT "Unit1.Em7.ControlNodes".cm.Command.jrWinderRearAxisY.posAbsolute[4] AND NOT "Unit1.Em7.ControlNodes".cm.Command.jrWinderRearAxisY.posAbsolute[5]);
END_REGION

REGION Network 177: CmJRWinderRearAxisY Position Absolute Position
   RUNG wire#powerrail
      Contact( "Unit1.Em7.ControlNodes".cm.Command.jrWinderRearAxisY.posAbsoluteSummary )
      Coil( "Unit1.Em7.ControlNodes".cmJRWinderRearAxisY.commands.posAbsolute )
   END_RUNG
   // the same network as SCL:
   "Unit1.Em7.ControlNodes".cmJRWinderRearAxisY.commands.posAbsolute := "Unit1.Em7.ControlNodes".cm.Command.jrWinderRearAxisY.posAbsoluteSummary;
END_REGION

REGION Network 178: CmJRWinderRearAxisY Interlock Summary
   RUNG wire#powerrail
      #instInterlockJRWinderRearAxisY(enableManualCmds := wire#w1, activeJobNumber :=, interlockSource := "Unit1.Em7.ControlNodes".cm.interlock.jrWinderRearAxisY.source, moduleInterface := "Unit1.Em7.HmiInterface".cmJRWinderRearAxisY, controlNode := "Unit1.Em7.ControlNodes".cmJRWinderRearAxisY, interlockcGeneral => "Unit1.Em7.ControlNodes".cm.interlock.jrWinderRearAxisY.permit.general)
   END_RUNG
   RUNG wire#powerrail
      I_Contact( #statUnitStatus.mode.production )
   END_RUNG wire#w1
   // the same network as SCL:
   #instInterlockJRWinderRearAxisY(enableManualCmds := NOT #statUnitStatus.mode.production,   // "LER_Axis64Pos_InterlockSummary"
                           interlockSource := "Unit1.Em7.ControlNodes".cm.interlock.jrWinderRearAxisY.source,
                           moduleInterface := "Unit1.Em7.HmiInterface".cmJRWinderRearAxisY,
                           controlNode := "Unit1.Em7.ControlNodes".cmJRWinderRearAxisY,
                           interlockcGeneral => "Unit1.Em7.ControlNodes".cm.interlock.jrWinderRearAxisY.permit.general);
END_REGION

REGION Network 179: CmJRWinderRearAxisY velocity/speed
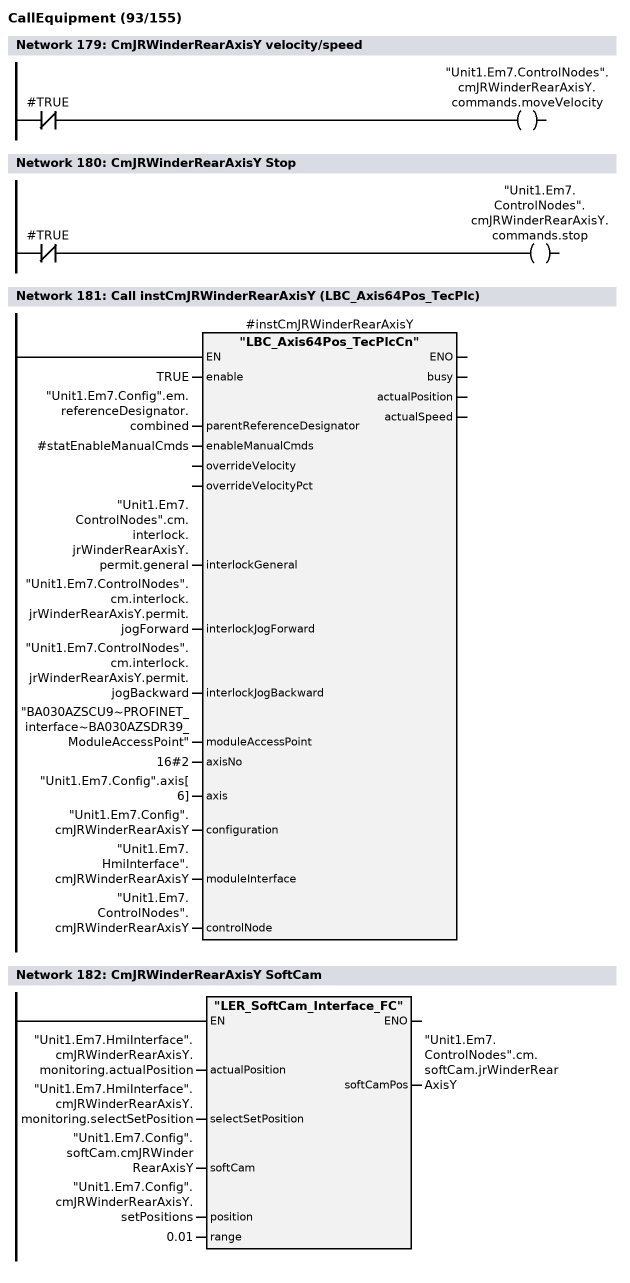
   RUNG wire#powerrail
      I_Contact( #TRUE )
      Coil( "Unit1.Em7.ControlNodes".cmJRWinderRearAxisY.commands.moveVelocity )
   END_RUNG
   // the same network as SCL:
   "Unit1.Em7.ControlNodes".cmJRWinderRearAxisY.commands.moveVelocity := NOT #TRUE;
END_REGION

REGION Network 180: CmJRWinderRearAxisY Stop
   RUNG wire#powerrail
      I_Contact( #TRUE )
      Coil( "Unit1.Em7.ControlNodes".cmJRWinderRearAxisY.commands.stop )
   END_RUNG
   // the same network as SCL:
   "Unit1.Em7.ControlNodes".cmJRWinderRearAxisY.commands.stop := NOT #TRUE;
END_REGION

REGION Network 181: Call instCmJRWinderRearAxisY (LBC_Axis64Pos_TecPlc)
   RUNG wire#powerrail
      #instCmJRWinderRearAxisY(enable := TRUE, parentReferenceDesignator := "Unit1.Em7.Config".em.referenceDesignator.combined, enableManualCmds := #statEnableManualCmds, overrideVelocity :=, overrideVelocityPct :=, interlockGeneral := "Unit1.Em7.ControlNodes".cm.interlock.jrWinderRearAxisY.permit.general, interlockJogForward := "Unit1.Em7.ControlNodes".cm.interlock.jrWinderRearAxisY.permit.jogForward, interlockJogBackward := "Unit1.Em7.ControlNodes".cm.interlock.jrWinderRearAxisY.permit.jogBackward, moduleAccessPoint := "BA030AZSCU9~PROFINET_interface~BA030AZSDR39_ModuleAccessPoint", axisNo := 16#2, axis := "Unit1.Em7.Config".axis[6], configuration := "Unit1.Em7.Config".cmJRWinderRearAxisY, moduleInterface := "Unit1.Em7.HmiInterface".cmJRWinderRearAxisY, controlNode := "Unit1.Em7.ControlNodes".cmJRWinderRearAxisY, busy =>, actualPosition =>, actualSpeed =>)
   END_RUNG
   // the same network as SCL:
   #instCmJRWinderRearAxisY(enable := TRUE,   // "LBC_Axis64Pos_TecPlcCn"
                           parentReferenceDesignator := "Unit1.Em7.Config".em.referenceDesignator.combined,
                           enableManualCmds := #statEnableManualCmds,
                           interlockGeneral := "Unit1.Em7.ControlNodes".cm.interlock.jrWinderRearAxisY.permit.general,
                           interlockJogForward := "Unit1.Em7.ControlNodes".cm.interlock.jrWinderRearAxisY.permit.jogForward,
                           interlockJogBackward := "Unit1.Em7.ControlNodes".cm.interlock.jrWinderRearAxisY.permit.jogBackward,
                           moduleAccessPoint := "BA030AZSCU9~PROFINET_interface~BA030AZSDR39_ModuleAccessPoint",
                           axisNo := 16#2,
                           axis := "Unit1.Em7.Config".axis[6],
                           configuration := "Unit1.Em7.Config".cmJRWinderRearAxisY,
                           moduleInterface := "Unit1.Em7.HmiInterface".cmJRWinderRearAxisY,
                           controlNode := "Unit1.Em7.ControlNodes".cmJRWinderRearAxisY);
END_REGION

REGION Network 182: CmJRWinderRearAxisY SoftCam
   RUNG wire#powerrail
      "LER_SoftCam_Interface_FC"(actualPosition := "Unit1.Em7.HmiInterface".cmJRWinderRearAxisY.monitoring.actualPosition, selectSetPosition := "Unit1.Em7.HmiInterface".cmJRWinderRearAxisY.monitoring.selectSetPosition, softCam := "Unit1.Em7.Config".softCam.cmJRWinderRearAxisY, position := "Unit1.Em7.Config".cmJRWinderRearAxisY.setPositions, range := 0.01, softCamPos => "Unit1.Em7.ControlNodes".cm.softCam.jrWinderRearAxisY)
   END_RUNG
   // the same network as SCL:
   "LER_SoftCam_Interface_FC"(actualPosition := "Unit1.Em7.HmiInterface".cmJRWinderRearAxisY.monitoring.actualPosition,
                           selectSetPosition := "Unit1.Em7.HmiInterface".cmJRWinderRearAxisY.monitoring.selectSetPosition,
                           softCam := "Unit1.Em7.Config".softCam.cmJRWinderRearAxisY,
                           position := "Unit1.Em7.Config".cmJRWinderRearAxisY.setPositions,
                           range := 0.01,
                           softCamPos => "Unit1.Em7.ControlNodes".cm.softCam.jrWinderRearAxisY);
END_REGION

REGION Network 184: JRWinderFrontAxisY Enable
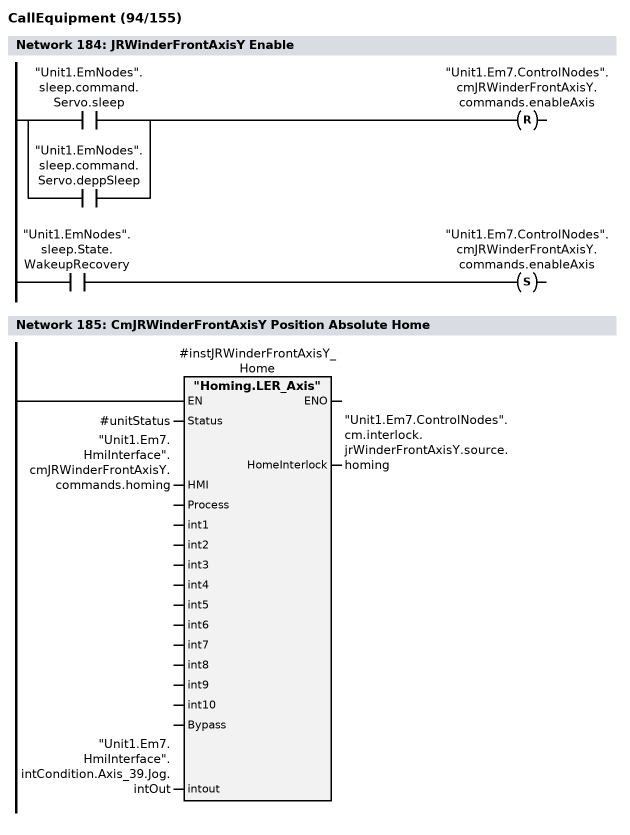
   RUNG wire#powerrail
      Contact( "Unit1.EmNodes".sleep.command.Servo.sleep )
      wire#w1
      R_Coil( "Unit1.Em7.ControlNodes".cmJRWinderFrontAxisY.commands.enableAxis )
   END_RUNG
   RUNG wire#powerrail
      Contact( "Unit1.EmNodes".sleep.command.Servo.deppSleep )
   END_RUNG wire#w1
   RUNG wire#powerrail
      Contact( "Unit1.EmNodes".sleep.State.WakeupRecovery )
      S_Coil( "Unit1.Em7.ControlNodes".cmJRWinderFrontAxisY.commands.enableAxis )
   END_RUNG
   // the same network as SCL:
   IF "Unit1.EmNodes".sleep.command.Servo.sleep OR "Unit1.EmNodes".sleep.command.Servo.deppSleep THEN
       "Unit1.Em7.ControlNodes".cmJRWinderFrontAxisY.commands.enableAxis := FALSE;
   END_IF;
   IF "Unit1.EmNodes".sleep.State.WakeupRecovery THEN
       "Unit1.Em7.ControlNodes".cmJRWinderFrontAxisY.commands.enableAxis := TRUE;
   END_IF;
END_REGION

REGION Network 185: CmJRWinderFrontAxisY Position Absolute Home
   RUNG wire#powerrail
      #instJRWinderFrontAxisY_Home(Status := #unitStatus, HMI := "Unit1.Em7.HmiInterface".cmJRWinderFrontAxisY.commands.homing, Process :=, int1 :=, int2 :=, int3 :=, int4 :=, int5 :=, int6 :=, int7 :=, int8 :=, int9 :=, int10 :=, Bypass :=, intout := "Unit1.Em7.HmiInterface".intCondition.Axis_39.Jog.intOut, HomeInterlock => "Unit1.Em7.ControlNodes".cm.interlock.jrWinderFrontAxisY.source.homing)
   END_RUNG
   // the same network as SCL:
   #instJRWinderFrontAxisY_Home(Status := #unitStatus,   // "Homing.LER_Axis"
                           HMI := "Unit1.Em7.HmiInterface".cmJRWinderFrontAxisY.commands.homing,
                           intout := "Unit1.Em7.HmiInterface".intCondition.Axis_39.Jog.intOut,
                           HomeInterlock => "Unit1.Em7.ControlNodes".cm.interlock.jrWinderFrontAxisY.source.homing);
END_REGION

REGION Network 186: CmJRWinderFrontAxisY Position Absolute Jog
